1500://判断负极叠台搬运是否有片，有片的话放到纠偏台
	IF NOT DP_SinStepe THEN
		IF CA_CarryingPos1  THEN//负极搬运、叠片各轴在初始位
			IF arrCyCtrl[arrCyNo.ElectValveName.CaDTCarryingVacuum].Io.DIOnSwitch AND  Mach_Control.Ca_b.Ca_DPCarryingFalg THEN//正极再取片位且叠台搬运有片,把当前片放到纠偏台
				DP_Step0:=1550;
			ELSE
				DP_Step0:=3000;	
			END_IF
		ELSE
			IF (Ca_Step0=0 OR Ca_Step0=6666) AND (Ca_Step3=0 OR Ca_Step3=6666) AND Scan_TON[2].Q THEN
				Scan_TON[2].IN:=FALSE;		
				DP_Step0:=9994;
				DTPosError[2]:=TRUE;
			END_IF
		END_IF
	END_IF	
1550://纠偏台回初始位
	//纠偏平台X1移动至初始位
	IF NOT DP_SinStepe THEN
		IF arrAxisCtrl[AxiseNo.AxisName.CadeviationX1].Status.Homed  AND arrAxisCtrl[AxiseNo.AxisName.CadeviationX1].Status.NoMoving AND NOT  arrAxisCtrl[AxiseNo.AxisName.CadeviationX1].Status.Error THEN
			IF arrAxisCtrl[AxiseNo.AxisName.CadeviationX1].Cmd.arrbRealPoint[1] THEN
				arrAxisCtrl[AxiseNo.AxisName.CadeviationX1].Cmd.iGoSetPos:=0;
			ELSE
				arrAxisCtrl[AxiseNo.AxisName.CadeviationX1].Cmd.iGoSetPos:=1;
			END_IF					
		END_IF
		//纠偏平台X2移动至初始位
		IF arrAxisCtrl[AxiseNo.AxisName.CadeviationX2].Status.Homed  AND arrAxisCtrl[AxiseNo.AxisName.CadeviationX2].Status.NoMoving AND NOT  arrAxisCtrl[AxiseNo.AxisName.CadeviationX2].Status.Error THEN
			IF arrAxisCtrl[AxiseNo.AxisName.CadeviationX2].Cmd.arrbRealPoint[1] THEN
				arrAxisCtrl[AxiseNo.AxisName.CadeviationX2].Cmd.iGoSetPos:=0;
			ELSE
				arrAxisCtrl[AxiseNo.AxisName.CadeviationX2].Cmd.iGoSetPos:=1;
			END_IF					
		END_IF
		//纠偏平台X2移动至初始位
		IF arrAxisCtrl[AxiseNo.AxisName.CadeviationY].Status.Homed  AND arrAxisCtrl[AxiseNo.AxisName.CadeviationY].Status.NoMoving AND NOT  arrAxisCtrl[AxiseNo.AxisName.CadeviationY].Status.Error THEN
			IF arrAxisCtrl[AxiseNo.AxisName.CadeviationY].Cmd.arrbRealPoint[1] THEN
				arrAxisCtrl[AxiseNo.AxisName.CadeviationY].Cmd.iGoSetPos:=0;
			ELSE
				arrAxisCtrl[AxiseNo.AxisName.CadeviationY].Cmd.iGoSetPos:=1;
			END_IF					
		END_IF
		IF arrAxisCtrl[AxiseNo.AxisName.CadeviationX1].Cmd.arrbRealPoint[1] AND arrAxisCtrl[AxiseNo.AxisName.CadeviationX2].Cmd.arrbRealPoint[1] AND arrAxisCtrl[AxiseNo.AxisName.CadeviationY].Cmd.arrbRealPoint[1] THEN
			DT_SingeMode();//单步选择	
			DP_Step0:=1600;	
			DT_TON[5].IN:=FALSE;
		END_IF	
	END_IF
1600:
	IF NOT DP_SinStepe THEN
		IF arrAxisCtrl[AxiseNo.AxisName.CaDTCarryingUpDown].Cmd.arrbRealPoint[3] THEN
			arrAxisCtrl[AxiseNo.AxisName.CaDTCarryingUpDown].Cmd.iGoSetPos:=0;
			/// 吸盘破真空    纠偏台开真空
			arrCyCtrl[arrCyNo.ElectValveName.CaDTCarryingVacuum].Cmd.bON:=TRUE;	//负极叠台搬运升降真空	真空
			arrCyCtrl[arrCyNo.ElectValveName.CaDTCarryingVacuum].Cmd.bOFF:=FALSE;	//负极叠台搬运升降真空破真空								
			arrCyCtrl[arrCyNo.ElectValveName.CadeviationVacuum].Cmd.bON:=TRUE;	//负极纠偏台真空			
			arrCyCtrl[arrCyNo.ElectValveName.CadeviationVacuum].Cmd.bOFF:=FALSE;	//负极纠偏台真空	   
			DT_SingeMode();//单步选择	
			DP_Step0:=1650;
			DT_TON[5].IN:=TRUE;
		ELSE
			arrAxisCtrl[AxiseNo.AxisName.CaDTCarryingUpDown].Cmd.iGoSetPos:=3;//负极搬运升降2上升至凸轮耦合初始高度
		END_IF	
	END_IF
1650://叠台搬运极片放回纠偏台
	IF NOT DP_SinStepe THEN
		 IF DT_TON[5].Q THEN
				IF arrAxisCtrl[AxiseNo.AxisName.CaDTCarryingUpDown].Cmd.arrbRealPoint[4] THEN
					arrAxisCtrl[AxiseNo.AxisName.CaDTCarryingUpDown].Cmd.iGoSetPos:=0;
					/// 吸盘破真空    纠偏台开真空
					Mach_Control.Ca_b.Ca_deviationFalg:=TRUE;//复位纠偏平台有料标记
					Mach_Control.Ca_b.Ca_DPCarryingFalg:=FALSE;//负极搬运真空吸盘有料标记复位
					Par.stDT_date.Ca_MQ_Slice[8]:=Par.stDT_date.Ca_MQ_Slice[9];
					DT_SingeMode();//单步选择	
					DP_Step0:=1700;
					DT_TON[5].IN:=FALSE;
				ELSE
					arrAxisCtrl[AxiseNo.AxisName.CaDTCarryingUpDown].Cmd.iGoSetPos:=4;//负极搬运升降2上升至凸轮耦合初始高度
				END_IF		
	    END_IF	
	END_IF	
1700:
	DP_Step0:=3000;	
	


	
2000:		
	IF NOT DP_SinStepe THEN
		IF AN_CarryingPos1  THEN//正极搬运、叠片各轴在初始位										
			IF CA_CarryingPos2 THEN//负极在叠片位
				IF arrAxisCtrl[AxiseNo.AxisName.SEPTATLine].Cmd.arrbRealPoint[1]  THEN
					IF Mach_Control.DT_b.SinStepMode THEN//单步调试模式
						DP_SinStepe:=TRUE;
					ELSE
						DP_SinStepe:=FALSE;	
					END_IF
					DP_Step0:=2010;//
				ELSE
					Mach_Control.DT_b.Error[6]:=TRUE;//叠正极片凸轮耦合时，隔膜平移轴即不在负极叠片位，也不在正极叠片位报警
					DP_Step0:=9998;
				END_IF;
			ELSIF  CA_CarryingPos1  THEN //负极取片位
				IF arrAxisCtrl[AxiseNo.AxisName.SEPTATLine].Cmd.arrbRealPoint[1]  THEN
					IF Mach_Control.DT_b.SinStepMode THEN//单步调试模式
						DP_SinStepe:=TRUE;
					ELSE
						DP_SinStepe:=FALSE;	
					END_IF
					DP_Step0:=2030;//
				ELSIF arrAxisCtrl[AxiseNo.AxisName.SEPTATLine].Cmd.arrbRealPoint[2]  THEN
					IF Mach_Control.DT_b.SinStepMode THEN//单步调试模式
						DP_SinStepe:=TRUE;
					ELSE
						DP_SinStepe:=FALSE;	
					END_IF
					DP_Step0:=2050;//
				ELSE
					Mach_Control.DT_b.Error[6]:=TRUE;//叠正极片凸轮耦合时，隔膜平移轴即不在负极叠片位，也不在正极叠片位报警
					DP_Step0:=9999;
				END_IF;							
			ELSE
				Mach_Control.DT_b.Error[7]:=TRUE;//叠正极片凸轮耦合时，负极取片即不在取片位，也不在叠片位
				DP_Step0:=10000;
			END_IF
		ELSE
			Mach_Control.DT_b.Error[8]:=TRUE;//叠正极片凸轮耦合时，正极片不在取片位
			DP_Step0:=10001;
		END_IF
	END_IF		


2010://负极搬运、叠片各轴在初始位，隔膜平移轴负极叠片位、正极叠片在放极片初始位
	IF NOT DP_SinStepe THEN
		An_CanIn5:=TRUE;
		IF Mach_Control.DT_b.SinStepMode THEN//单步调试模式
				DP_SinStepe:=TRUE;
			ELSE
				DP_SinStepe:=FALSE;	
			END_IF
		DP_Step0:=2020;	
	END_IF	
2020:
	IF NOT DP_SinStepe THEN
		IF NOT An_CanIn5 THEN
			IF Mach_Control.DT_b.SinStepMode THEN//单步调试模式
				DP_SinStepe:=TRUE;
			ELSE
				DP_SinStepe:=FALSE;	
			END_IF	
			DP_Step0:=2070;
		ELSIF fbAnCamInCarryingLine.bError  OR fbAnCamInDTCarryingLine.bError OR fbAnCamInDTCarryingUpDown.bError OR 
			fbAnCamInCarryingWhirling.bError OR fbCaCamInCarryingLine2.bError OR 
			fbCaCamInDTCarryingUpDown.bError OR fbCamInGMBuffer.bError OR fbCamInGMDanserMove.bError OR fbCamInVirGMDriver.bError   OR
			fbCamInRightYDUpDown.bError OR fbCamInRightYDLine.bError  THEN
			An_CanIn5:=FALSE;
			Mach_Control.DT_b.Error[19]:=TRUE;//凸轮耦合报警
			DP_Step0:=10004;		
		END_IF
	END_IF		
2030://负极搬运、叠片各轴在初始位，隔膜平移轴负极叠片位、正极叠片在取极片位
	IF NOT DP_SinStepe THEN
		IF Mach_Control.DT_b.SinStepMode THEN//单步调试模式
			DP_SinStepe:=TRUE;
		ELSE
			DP_SinStepe:=FALSE;	
		END_IF
		An_CanIn6:=TRUE;
		DP_Step0:=2040;
	END_IF
2040:
	IF NOT DP_SinStepe THEN
		IF NOT An_CanIn6 THEN
			IF Mach_Control.DT_b.SinStepMode THEN//单步调试模式
				DP_SinStepe:=TRUE;
			ELSE
				DP_SinStepe:=FALSE;	
			END_IF
			DP_Step0:=2070;
		ELSIF fbAnCamInCarryingLine.bError OR fbAnCamInDTCarryingLine.bError OR
			fbAnCamInDTCarryingUpDown.bError OR fbAnCamInCarryingWhirling.bError OR fbCamInGMBuffer.bError OR
			fbCamInGMDanserMove.bError OR fbCamInVirGMDriver.bError  OR fbCamInRightYDUpDown.bError OR
			fbCamInRightYDLine.bError  THEN
			An_CanIn6:=FALSE;
			Mach_Control.DT_b.Error[19]:=TRUE;//凸轮耦合报警
			DP_Step0:=10002;									
		END_IF
	END_IF
2050://负极搬运、叠片各轴在初始位，隔膜平移轴正极叠片位、正极叠片在取极片位
	IF NOT DP_SinStepe THEN
		An_CanIn7:=TRUE;
		IF Mach_Control.DT_b.SinStepMode THEN//单步调试模式
				DP_SinStepe:=TRUE;
			ELSE
				DP_SinStepe:=FALSE;	
			END_IF
		DP_Step0:=2060;
	END_IF
2060:
	IF NOT DP_SinStepe THEN
			arrAxisCtrl[AxiseNo.VirAxisName.VirMain].Cmd	.bMoveAbs:=FALSE;	
			IF NOT An_CanIn7 THEN
				IF Mach_Control.DT_b.SinStepMode THEN//单步调试模式
					DP_SinStepe:=TRUE;
				ELSE
					DP_SinStepe:=FALSE;	
				END_IF
				DP_Step0:=2070;
			ELSIF fbAnCamInCarryingLine.bError OR fbAnCamInCarryingUpDown.bError OR fbAnCamInDTCarryingLine.bError OR fbAnCamInDTCarryingUpDown.bError OR 
				fbAnCamInCarryingWhirling.bError OR fbCamInRightYDUpDown.bError OR fbCamInRightYDLine.bError THEN
				An_CanIn7:=FALSE;
				Mach_Control.DT_b.Error[19]:=TRUE;//凸轮耦合报警
				DP_Step0:=10003;												
			END_IF
	END_IF	
	
2070://判断正极叠片搬运机械手上是否有极片

	IF NOT DP_SinStepe THEN
		VirMain_TON.IN:=FALSE;
		IF (NOT arrCyCtrl[arrCyNo.ElectValveName.AnDTCarryingVacuum].Io.DIOnSwitch AND NOT Mach_Control.An_b.An_DPCarryingFalg) OR Bnt_Blueflaging THEN	
			IF Mach_Control.DT_b.SinStepMode THEN//单步调试模式
				DP_SinStepe:=TRUE;
			ELSE
				DP_SinStepe:=FALSE;	
			END_IF
			DP_Step0:=2071;
		ELSE	
		  	Mach_Control.An_b.Error[28]:=TRUE; //正极叠片完空叠隔膜时，正极叠片搬运机械手真空有信号、标记有极片报警,请拿掉极片
		END_IF  
	END_IF

2071://主轴启动
	IF NOT DP_SinStepe THEN
		arrAxisCtrl[AxiseNo.VirAxisName.VirMain].Cmd	.bDynamitcsParSel:=2;	
		arrAxisPar[AxiseNo.VirAxisName.VirMain].fTagatTime:=VirMain_TagatTime;
		arrAxisCtrl[AxiseNo.VirAxisName.VirMain].Cmd	.fPositon_of_Abs:=360;
		arrAxisCtrl[AxiseNo.VirAxisName.VirMain].Cmd	.bMoveAbs:=TRUE;	
		//fbCaCamInCarryingUpDown2OutCamFlge:=FALSE;//负极升降2凸轮解耦标记										
		IF  arrAxis[AxiseNo.VirAxisName.VirMain].Status.Moving OR arrAxisCtrl[AxiseNo.VirAxisName.VirMain].Status.fActPos>=10  THEN
			VirMain_TON.IN:=FALSE;
			arrAxisCtrl[AxiseNo.VirAxisName.VirMain].Cmd	.bMoveAbs:=FALSE;	
			DP_Step0:=2080;	
		ELSE
			IF NOT VirMain_TON.Q THEN
				VirMain_TON.IN:=TRUE;
			ELSE
				VirMain_TON.IN:=FALSE;
				Mach_Control.DT_b.Error[22]:=TRUE;//主轴启动超时报警
				DP_Step0:=10006;	
			END_IF	
		END_IF	
	END_IF				
			
(*2080:
IF arrAxis[AxiseNo.VirAxisName.VirMain].NcToPlc.SetPos>=234 AND arrAxis[AxiseNo.VirAxisName.VirMain].NcToPlc.SetPos<=240 THEN
	arrCyCtrl[arrCyNo.ElectValveName.AnDTCarryingVacuum].Cmd.bOFF:=TRUE;//正极叠片搬运真空关
	arrCyCtrl[arrCyNo.ElectValveName.AnDTCarryingVacuumBark].Cmd.bON:=TRUE;//正极叠片搬运破真空开
	Mach_Control.An_b.An_DPCarryingFalg :=FALSE;//复位正极叠片搬运吸盘上有料标记																									
END_IF				
IF arrAxis[AxiseNo.VirAxisName.VirMain].NcToPlc.SetPos=360 AND  arrAxis[AxiseNo.VirAxisName.VirMain].Status.NotMoving  THEN
			Mach_Control.An_b.An_KDQuantited:=Mach_Control.An_b.An_KDQuantited +1;
			DP_Step1:=100;//解除耦合，主轴回零子程序
			arrAxisCtrl[AxiseNo.AxisName.DTUpDown].Cmd.fPosition_of_Rel:=-Par.stDT_date.SEPTA_Thickness;
			arrAxisPar[AxiseNo.AxisName.DTUpDown].fVelocity_of_Rel:=100;
			arrAxisCtrl[AxiseNo.AxisName.DTUpDown].Cmd.bMoveRel:=TRUE;
			DP_Step0:=0;
END_IF*)

3000:
	IF NOT DP_SinStepe THEN		
		Scan_TON[2].IN:=TRUE;	
		IF CA_CarryingPos1  THEN//负极搬运、叠片各轴在初始位
			Scan_TON[1].IN:=TRUE;	
			IF AN_CarryingPos2  THEN//正极在叠片位	
				IF arrAxisCtrl[AxiseNo.AxisName.SEPTATLine].Cmd.arrbRealPoint[2]   THEN													
					IF Mach_Control.DT_b.SinStepMode THEN//单步调试模式
						DP_SinStepe:=TRUE;
					ELSE
						DP_SinStepe:=FALSE;	
					END_IF												
					DP_Step0:=3010;//													
				ELSE
					Mach_Control.DT_b.Error[5]:=TRUE;//叠负极片凸轮耦合时，隔膜平移轴即不在负极叠片位，也不在正极叠片位报警
					DP_Step0:=9991;	
				END_IF;
			ELSIF AN_CarryingPos1  THEN//在取片位																		
				IF arrAxisCtrl[AxiseNo.AxisName.SEPTATLine].Cmd.arrbRealPoint[1]  THEN
					IF Mach_Control.DT_b.SinStepMode THEN//单步调试模式
						DP_SinStepe:=TRUE;
					ELSE
						DP_SinStepe:=FALSE;	
					END_IF											
					DP_Step0:=3030;//
				ELSIF arrAxisCtrl[AxiseNo.AxisName.SEPTATLine].Cmd.arrbRealPoint[2] THEN
					IF Mach_Control.DT_b.SinStepMode THEN//单步调试模式
						DP_SinStepe:=TRUE;
					ELSE
						DP_SinStepe:=FALSE;	
					END_IF											
					DP_Step0:=3050;//
				ELSE
					Mach_Control.DT_b.Error[5]:=TRUE;//叠负极片凸轮耦合时，隔膜平移轴即不在负极叠片位，也不在正极叠片位报警
					DP_Step0:=9992;	
				END_IF;							
			ELSIF Scan_TON[1].Q THEN
				Scan_TON[1].IN:=FALSE;	
				DP_Step0:=9993;
				DTPosError[4]:=TRUE;
			END_IF
		ELSE
			IF (Ca_Step0=0 OR Ca_Step0=6666) AND (Ca_Step3=0 OR Ca_Step3=6666) AND Scan_TON[2].Q THEN
				Scan_TON[2].IN:=FALSE;		
				DP_Step0:=9994;
				DTPosError[2]:=TRUE;
			END_IF
		END_IF
END_IF		

3010://负极搬运、叠片各轴在初始位，隔膜平移轴正极叠片位、正极叠片在放极片初始位
	IF NOT DP_SinStepe THEN
		Ca_CanIn5:=TRUE;
		IF Mach_Control.DT_b.SinStepMode THEN//单步调试模式
			DP_SinStepe:=TRUE;
		ELSE
			DP_SinStepe:=FALSE;	
		END_IF
		DP_Step0:=3020;	
	END_IF
3020:
	IF NOT DP_SinStepe THEN
		arrAxisCtrl[AxiseNo.VirAxisName.VirMain].Cmd	.bMoveAbs:=FALSE;	
		IF NOT Ca_CanIn5 THEN
			IF Mach_Control.DT_b.SinStepMode THEN//单步调试模式
				DP_SinStepe:=TRUE;
			ELSE
				DP_SinStepe:=FALSE;	
			END_IF
			DP_Step0:=3070;	
		ELSIF fbCaCamInCarryingLine2.bError OR  fbCaCamInDTCarryingLine.bError OR fbCaCamInDTCarryingUpDown.bError OR 
			fbCamInGMBuffer.bError OR fbCamInGMDanserMove.bError OR fbCamInVirGMDriver.bError OR fbAnCamInCarryingLine.bError OR 
			fbAnCamInDTCarryingLine.bError OR fbAnCamInCarryingWhirling.bError OR fbCamInLeftYDUpDown.bError OR fbCamInLeftYDLine.bError THEN
			Ca_CanIn5:=FALSE;
			Mach_Control.DT_b.Error[19]:=TRUE;//凸轮耦合报警
			DP_Step0:=9998;										
		END_IF
	END_IF
3030://负极搬运、叠片各轴在初始位，隔膜平移轴负极叠片位、正极叠片在取极片位
	IF NOT DP_SinStepe THEN
		Ca_CanIn6:=TRUE;
		IF Mach_Control.DT_b.SinStepMode THEN//单步调试模式
			DP_SinStepe:=TRUE;
		ELSE
			DP_SinStepe:=FALSE;	
		END_IF
		DP_Step0:=3040;
	END_IF
3040://判断凸轮耦合是否完成
	IF NOT DP_SinStepe THEN
		IF NOT Ca_CanIn6 THEN
			IF Mach_Control.DT_b.SinStepMode THEN//单步调试模式
				DP_SinStepe:=TRUE;
			ELSE
				DP_SinStepe:=FALSE;	
			END_IF
			DP_Step0:=3070;
		ELSIF  fbCaCamInCarryingLine2.bError OR fbCaCamInDTCarryingLine.bError OR 
			fbCaCamInDTCarryingUpDown.bError OR fbCamInLeftYDUpDown.bError OR 	fbCamInLeftYDLine.bError THEN										
			Ca_CanIn6:=FALSE;
			Mach_Control.DT_b.Error[19]:=TRUE;//凸轮耦合报警
			DP_Step0:=9995;		
		END_IF
	END_IF
3050://负极搬运、叠片各轴在初始位，隔膜平移轴正极叠片位、正极叠片在取极片位
	IF NOT DP_SinStepe THEN
		Ca_CanIn7:=TRUE;
		IF Mach_Control.DT_b.SinStepMode THEN//单步调试模式
			DP_SinStepe:=TRUE;
		ELSE
			DP_SinStepe:=FALSE;	
		END_IF
		DP_Step0:=3060;
	END_IF
3060:
	IF NOT DP_SinStepe THEN
			arrAxisCtrl[AxiseNo.VirAxisName.VirMain].Cmd	.bMoveAbs:=FALSE;	
			IF NOT Ca_CanIn7 THEN
				IF Mach_Control.DT_b.SinStepMode THEN//单步调试模式
					DP_SinStepe:=TRUE;
				ELSE
					DP_SinStepe:=FALSE;	
				END_IF																			
				DP_Step0:=3070;
			ELSIF fbCaCamInCarryingLine2.bError OR fbCaCamInDTCarryingLine.bError OR 
				fbCaCamInDTCarryingUpDown.bError OR fbCamInGMBuffer.bError OR fbCamInGMDanserMove.bError OR
				fbCamInVirGMDriver.bError OR fbCamInLeftYDUpDown.bError OR fbCamInLeftYDLine.bError  THEN
				Ca_CanIn7:=FALSE;
				Mach_Control.DT_b.Error[19]:=TRUE;//凸轮耦合报警
				DP_Step0:=9996;	
			END_IF
	END_IF

3070://判断负极叠片搬运机械手上是否有极片
	VirMain_TON.IN:=FALSE;
	DP_Step0:=3071;
	(*
	IF NOT DP_SinStepe THEN
		IF NOT arrCyCtrl[arrCyNo.ElectValveName.CaDTCarryingVacuum].Io.DIOnSwitch AND NOT Mach_Control.Ca_b.Ca_DPCarryingFalg  THEN	
			IF Mach_Control.DT_b.SinStepMode THEN//单步调试模式
				DP_SinStepe:=TRUE;
			ELSE
				DP_SinStepe:=FALSE;	
			END_IF
			DP_Step0:=3071;
		ELSE	
		  	Mach_Control.Ca_b.Error[28]:=TRUE; //负极叠片完空叠隔膜时，负极叠片搬运机械手真空检测有信号报警,请拿掉极片
		END_IF  
	END_IF	 
	*)
3071://主轴启动
	IF NOT DP_SinStepe THEN
		arrAxisCtrl[AxiseNo.VirAxisName.VirMain].Cmd	.bDynamitcsParSel:=2;
		arrAxisPar[AxiseNo.VirAxisName.VirMain].fTagatTime:=VirMain_TagatTime;
		arrAxisCtrl[AxiseNo.VirAxisName.VirMain].Cmd	.fPositon_of_Abs:=360;
		arrAxisCtrl[AxiseNo.VirAxisName.VirMain].Cmd	.bMoveAbs:=TRUE;	
		//fbCaCamInCarryingUpDown2OutCamFlge:=FALSE;//负极升降2凸轮解耦标记										
		IF  arrAxis[AxiseNo.VirAxisName.VirMain].Status.Moving OR arrAxisCtrl[AxiseNo.VirAxisName.VirMain].Status.fActPos>=10  THEN
			VirMain_TON.IN:=FALSE;
			arrAxisCtrl[AxiseNo.VirAxisName.VirMain].Cmd	.bMoveAbs:=FALSE;	
			DP_Step0:=3080;	
		ELSE
			IF NOT VirMain_TON.Q THEN
				VirMain_TON.IN:=TRUE;
			ELSE
				VirMain_TON.IN:=FALSE;
				Mach_Control.DT_b.Error[22]:=TRUE;//主轴启动超时报警
				DP_Step0:=10006;	
			END_IF	
		END_IF	
	END_IF	

END_CASE
END_IF


(**************************************************************************************电芯下料**************************************************************************************************************)
CASE DP_Step0 OF
2080:
IF arrAxis[AxiseNo.VirAxisName.VirMain].NcToPlc.SetPos>=234 AND arrAxis[AxiseNo.VirAxisName.VirMain].NcToPlc.SetPos<=240 THEN
	arrCyCtrl[arrCyNo.ElectValveName.AnDTCarryingVacuum].Cmd.bOFF:=FALSE;//正极叠片搬运升降真空关
     arrCyCtrl[arrCyNo.ElectValveName.AnDTCarryingVacuum].Cmd.bON:=TRUE;//正极叠片搬运升降真空关
	Mach_Control.An_b.An_DPCarryingFalg :=FALSE;//复位正极叠片搬运吸盘上有料标记																									
END_IF				
IF arrAxis[AxiseNo.VirAxisName.VirMain].NcToPlc.SetPos=360 AND  arrAxis[AxiseNo.VirAxisName.VirMain].Status.NotMoving  THEN
			Mach_Control.An_b.An_KDQuantited:=Mach_Control.An_b.An_KDQuantited +1;
			DP_Step1:=100;//解除耦合，主轴回零子程序
			arrAxisCtrl[AxiseNo.AxisName.DTUpDown].Cmd.fPosition_of_Rel:=-Par.stDT_date.SEPTA_Thickness;
			arrAxisPar[AxiseNo.AxisName.DTUpDown].fVelocity_of_Rel:=100;
			arrAxisCtrl[AxiseNo.AxisName.DTUpDown].Cmd.bMoveRel:=TRUE;
			DP_Step0:=0;
END_IF
	
(*2080:
	IF arrAxis[AxiseNo.VirAxisName.VirMain].NcToPlc.SetPos=360 AND  arrAxis[AxiseNo.VirAxisName.VirMain].Status.NotMoving  THEN
		Mach_Control.An_b.An_KDQuantited:=Mach_Control.An_b.An_KDQuantited +1;
		DPcount:=DPcount+1;	
		DP_Step1:=100;//解除耦合，主轴回零子程序
		arrAxisCtrl[AxiseNo.AxisName.DTUpDown].Cmd.fPosition_of_Rel:=-Par.stDT_date.SEPTA_Thickness;
		arrAxisPar[AxiseNo.AxisName.DTUpDown].fVelocity_of_Rel:=100;
		arrAxisCtrl[AxiseNo.AxisName.DTUpDown].Cmd.bMoveRel:=TRUE;
		DP_Step0:=0;
	END_IF*)


3080:

	IF arrAxis[AxiseNo.VirAxisName.VirMain].NcToPlc.SetPos=360 AND  arrAxis[AxiseNo.VirAxisName.VirMain].Status.NotMoving  THEN
		Mach_Control.Ca_b.Ca_KDQuantited:=Mach_Control.Ca_b.Ca_KDQuantited +1;
		DPcount:=DPcount+1;	
		DP_Step1:=100;//解除耦合，主轴回零子程序
		arrAxisCtrl[AxiseNo.AxisName.DTUpDown].Cmd.fPosition_of_Rel:=-Par.stDT_date.SEPTA_Thickness;
		arrAxisPar[AxiseNo.AxisName.DTUpDown].fVelocity_of_Rel:=100;
		arrAxisCtrl[AxiseNo.AxisName.DTUpDown].Cmd.bMoveRel:=TRUE;							
		DP_Step0:=0;
	END_IF		
END_CASE
END_ACTION

ACTION _01DT_Auto4:
IF Mach_Control.U.DT_iMode=1 THEN//在自动状态下
CASE DP_Step0 OF		
	6000://叠片完成，负极升降机械手回到安全位
			IF NOT DP_SinStepe THEN
						//负极取片2升降安全位
						IF arrAxisCtrl[AxiseNo.AxisName.CaCarryingUpDown2].Status.Homed AND arrAxisCtrl[AxiseNo.AxisName.CaCarryingUpDown2].Status.NoMoving AND 
							NOT arrAxisCtrl[AxiseNo.AxisName.CaCarryingUpDown2].Status.Error THEN
								IF arrAxisCtrl[AxiseNo.AxisName.CaCarryingUpDown2].Cmd.arrbRealPoint[4] THEN
										arrAxisCtrl[AxiseNo.AxisName.CaCarryingUpDown2].Cmd.iGoSetPos:=0;
								ELSE
									arrAxisCtrl[AxiseNo.AxisName.CaCarryingUpDown2].Cmd.iGoSetPos:=4;//负极搬运升降2移动至初始高度
								END_IF
						END_IF				
						//负极叠片取片升降等待位
						IF arrAxisCtrl[AxiseNo.AxisName.CaDTCarryingUpDown].Status.Homed AND arrAxisCtrl[AxiseNo.AxisName.CaDTCarryingUpDown].Status.NoMoving AND
							 NOT arrAxisCtrl[AxiseNo.AxisName.CaDTCarryingUpDown].Status.Error THEN
									IF arrAxisCtrl[AxiseNo.AxisName.CaDTCarryingUpDown].Cmd.arrbRealPoint[4] THEN
											arrAxisCtrl[AxiseNo.AxisName.CaDTCarryingUpDown].Cmd.iGoSetPos:=0;							
									ELSE
										arrAxisCtrl[AxiseNo.AxisName.CaDTCarryingUpDown].Cmd.iGoSetPos:=4;//负极叠片升降移动至等待高度
									END_IF
						END_IF
						
						IF 	arrAxisCtrl[AxiseNo.AxisName.CaCarryingUpDown2].Cmd.arrbRealPoint[4]  AND  arrAxisCtrl[AxiseNo.AxisName.CaCarryingUpDown2].Status.NoMoving AND 
								arrAxisCtrl[AxiseNo.AxisName.CaDTCarryingUpDown].Cmd.arrbRealPoint[4] 	AND arrAxisCtrl[AxiseNo.AxisName.CaDTCarryingUpDown].Status.NoMoving THEN
								IF Mach_Control.DT_b.SinStepMode THEN//单步调试模式
											DP_SinStepe:=TRUE;
								ELSE
											DP_SinStepe:=FALSE;	
								END_IF
								DP_Step0:=6010;
					END_IF
			END_IF
		6010://判断主轴是否停止、是否在初始位、是否有轴在耦合中
			IF NOT DP_SinStepe THEN
				IF CA_CarryingPos2 THEN
					IF arrAxisCtrl[AxiseNo.VirAxisName.VirMain].Status.NoMoving AND arrAxis[AxiseNo.VirAxisName.VirMain].NcToPlc.ActPos=0 AND NOT DT_AxiseCoupling THEN
						DT_SingeMode();//单步选择						
						DP_Step0:=6012;
					ELSE
						DP_Step1:=100;//调用主轴回初始位子程序
						DT_SingeMode();//单步选择							
						DP_Step0:=6011;
					END_IF
				ELSIF  CA_CarryingPos1 THEN
					DP_Step0:=6014;
				END_IF	
			END_IF
					
		6011://判断主轴的模长的当前位置是否为0
			IF NOT DP_SinStepe THEN
				IF DP_Step1=6666 AND arrAxisCtrl[AxiseNo.VirAxisName.VirMain].Status.NoMoving AND arrAxis[AxiseNo.VirAxisName.VirMain].NcToPlc.ActPos=0 AND NOT DT_AxiseCoupling THEN
					DT_SingeMode();//单步选择						
					DP_Step0:=6012;
				END_IF
			END_IF		

		6012:
			//负极送片搬运平移
				fbCaCamInCarryingLine2.ParCamIn.SlaveScaling:=-1;
				fbCaCamInCarryingLine2.bCamInExecute:=TRUE;								
		        fbCaCamInCarryingUpDown2.iTableSel:=3;    //20240528SJ
	            fbCaCamInCarryingUpDown2.bCamInExecute:=TRUE;		
				
			//负极叠台搬运平移
				fbCaCamInDTCarryingLine.ParCamIn.SlaveScaling:=-1;
				fbCaCamInDTCarryingLine.bCamInExecute:=TRUE;	
			    fbCaCamInDTCarryingUpDown.iTableSel:=3;   //20240528SJ
	            fbCaCamInDTCarryingUpDown.bCamInExecute:=TRUE;
				
			//负极叠片升降轴放片凸轮耦合
				//fbCaCamInDTCarryingUpDown.iTableSel:=2;
				//fbCaCamInDTCarryingUpDown.bCamInExecute:=TRUE;		
														  
			IF fbCaCamInCarryingLine2.bInSync AND fbCaCamInDTCarryingLine.bInSync AND  fbCaCamInCarryingUpDown2.bInSync AND fbCaCamInDTCarryingUpDown.bInSync   THEN   
				DT_SingeMode();//单步选择		
				DP_Step0:=6013;
			ELSIF fbCaCamInCarryingLine2.bError  OR  fbCaCamInDTCarryingLine.bError  OR 
                    fbCaCamInCarryingUpDown2.bError OR fbCaCamInDTCarryingUpDown.bError   THEN   
				Mach_Control.DT_b.Error[19]:=TRUE;//凸轮耦合报警
			END_IF	
		6074:	
			IF arrAxis[AxiseNo.VirAxisName.VirMain].NcToPlc.SetPos=360 AND  arrAxis[AxiseNo.VirAxisName.VirMain].Status.NotMoving THEN 
				DP_Step1:=100;
				DP_Step0:=6075;	
			END_IF
		  
		6075:  
			IF DP_Step1=6666 THEN	
				DP_Step0:=6014;						
			END_IF		
		  
		6014:
			IF arrAxisCtrl[AxiseNo.VirAxisName.VirMain].Status.NoMoving AND arrAxis[AxiseNo.VirAxisName.VirMain].NcToPlc.ActPos=0 AND NOT DT_AxiseCoupling 
				AND CA_CarryingPos1 THEN
				DP_Step0:=6015;	
			ELSIF  DT_AxiseCoupling THEN
				DP_Step1:=100;
				DP_Step0:=6075;	
			END_IF  
	(*
				IF NOT DP_SinStepe THEN
					//负极取片2平移取片位
											IF arrAxisCtrl[AxiseNo.AxisName.CaCarryingUpDown2].Cmd.arrbRealPoint[5] AND arrAxisCtrl[AxiseNo.AxisName.CaCarryingLine2].Status.Homed AND
												 arrAxisCtrl[AxiseNo.AxisName.CaCarryingLine2].Status.NoMoving AND NOT arrAxisCtrl[AxiseNo.AxisName.CaCarryingLine2].Status.Error THEN
													IF arrAxisCtrl[AxiseNo.AxisName.CaCarryingLine2].Cmd.arrbRealPoint[1] THEN
															arrAxisCtrl[AxiseNo.AxisName.CaCarryingLine2].Cmd.iGoSetPos:=0;					
													ELSE
														arrAxisCtrl[AxiseNo.AxisName.CaCarryingLine2].Cmd.iGoSetPos:=1;//负极搬运平移2移动至初始位取流水线上的极片
													END_IF
											END_IF
					//负极叠片平移取片位
										IF TailCurlSEPTA_SafePos  AND arrAxisCtrl[AxiseNo.AxisName.CaDTCarryingUpDown].Cmd.arrbRealPoint[4] AND arrAxisCtrl[AxiseNo.AxisName.CaDTCarryingLine].Status.Homed AND
											 arrAxisCtrl[AxiseNo.AxisName.CaDTCarryingLine].Status.NoMoving AND NOT arrAxisCtrl[AxiseNo.AxisName.CaDTCarryingLine].Status.Error THEN
												IF arrAxisCtrl[AxiseNo.AxisName.CaDTCarryingLine].Cmd.arrbRealPoint[1] THEN
														arrAxisCtrl[AxiseNo.AxisName.CaDTCarryingLine].Cmd.iGoSetPos:=0;
												ELSE
													arrAxisCtrl[AxiseNo.AxisName.CaDTCarryingLine].Cmd.iGoSetPos:=1;//负极叠片平移至初始位
												END_IF
										END_IF
										
										IF 	arrAxisCtrl[AxiseNo.AxisName.CaCarryingLine2].Cmd.arrbRealPoint[1] AND 	arrAxisCtrl[AxiseNo.AxisName.CaCarryingLine2].Status.NoMoving AND 
													arrAxisCtrl[AxiseNo.AxisName.CaDTCarryingLine].Cmd.arrbRealPoint[1] AND 	arrAxisCtrl[AxiseNo.AxisName.CaDTCarryingLine].Status.NoMoving THEN
													IF Mach_Control.DT_b.SinStepMode THEN//单步调试模式
																DP_SinStepe:=TRUE;
													ELSE
																DP_SinStepe:=FALSE;	
													END_IF
													DP_Step0:=6015;	
										//ELSIF  THEN											
										END_IF
				END_IF
	*)			
		6015:
			IF NOT DP_SinStepe THEN
					//负极叠片升降避让位
					IF arrAxisCtrl[AxiseNo.AxisName.CaDTCarryingUpDown].Status.Homed AND arrAxisCtrl[AxiseNo.AxisName.CaDTCarryingUpDown].Status.NoMoving AND
						 NOT arrAxisCtrl[AxiseNo.AxisName.CaDTCarryingUpDown].Status.Error THEN
						IF arrAxisCtrl[AxiseNo.AxisName.CaDTCarryingUpDown].Cmd.arrbRealPoint[5] THEN
								arrAxisCtrl[AxiseNo.AxisName.CaDTCarryingUpDown].Cmd.iGoSetPos:=0;							
						ELSE
							arrAxisCtrl[AxiseNo.AxisName.CaDTCarryingUpDown].Cmd.iGoSetPos:=5;//负极叠片升降移动至避让高度
						END_IF
					END_IF
					
					IF 	arrAxisCtrl[AxiseNo.AxisName.CaDTCarryingUpDown].Cmd.arrbRealPoint[5] 	AND arrAxisCtrl[AxiseNo.AxisName.CaDTCarryingUpDown].Status.NoMoving THEN
						IF Mach_Control.DT_b.SinStepMode THEN//单步调试模式
							DP_SinStepe:=TRUE;
						ELSE
							DP_SinStepe:=FALSE;	
						END_IF
						DP_Step0:=6016;
				END_IF
			END_IF
END_CASE
END_IF


CASE DP_Step0 OF
	6013:
		IF NOT DP_SinStepe THEN
			 arrAxisCtrl[AxiseNo.VirAxisName.VirMain].Cmd.bDynamitcsParSel:=2;	
			 arrAxisPar[AxiseNo.VirAxisName.VirMain].fTagatTime:=VirMain_TagatTime;
			 arrAxisCtrl[AxiseNo.VirAxisName.VirMain].Cmd.fPositon_of_Abs:=360;
			 arrAxisCtrl[AxiseNo.VirAxisName.VirMain].Cmd.bMoveAbs:=TRUE;			
			IF  arrAxis[AxiseNo.VirAxisName.VirMain].Status.Moving OR arrAxisCtrl[AxiseNo.VirAxisName.VirMain].Status.fActPos>=5  THEN		
				arrAxisCtrl[AxiseNo.VirAxisName.VirMain].Cmd.bMoveAbs:=FALSE;
				Ca_TON[2].IN:=FALSE;                               	
				DP_Step0:=6074;	
				//Ca_StandbyStep1:=300;  //取消调用负极送片搬运取流水线极片
				//Ca_StandbyStep5:=400;
			ELSE
				IF NOT Ca_TON[2].Q THEN
					Ca_TON[2].IN:=TRUE;
				ELSE
				Ca_TON[2].IN:=FALSE;
					Mach_Control.DT_b.Error[22]:=TRUE;//主轴启动超时报警
					arrAxisCtrl[AxiseNo.VirAxisName.VirMain].Cmd	.bMoveAbs:=FALSE;	
				END_IF
			END_IF	
		END_IF	
					
	6016://纠偏平台回原
		 IF arrAxisCtrl[AxiseNo.AxisName.AnDTCarryingUpDown].Cmd.arrbRealPoint[4] AND arrAxisCtrl[AxiseNo.AxisName.CaDTCarryingUpDown].Cmd.arrbRealPoint[5]  THEN
			 DP_Step11:=100;//正极纠偏平台回原
			 DP_Step12:=100;//负极纠偏平台回原
			 DP_Step0:=6020;
		 END_IF


	6020:
				IF Mach_Control.DT_b.DT_Oerhang_Z<>2 OR   Mach_Control.DT_b.DT_Overhang THEN
					CellMemory[Mach_Control.DT_b.DT_Memory].Hough:=1;
					DP_Step0:=6025;
					NN:=0;
				ELSE 
					CellMemory[Mach_Control.DT_b.DT_Memory].Hough:=2;
					DP_Step0:=6024;
				END_IF
				
	6024:
				NN:=NN+1;
				DP_Step0:=6025;			
																
	6025:
			Mach_Control.DT_b.DT_amount:=Mach_Control.DT_b.DT_amount+1;
			CellMemory[Mach_Control.DT_b.DT_Memory].Cell:=TRUE;	
			CellMemory[Mach_Control.DT_b.DT_Memory].DT_station_No:=Mach_Control.DT_b.DT_No;
			CellMemory[Mach_Control.DT_b.DT_Memory].DT_speed:=Par.stDT_date.SinglePosTime;
			CellMemory[Mach_Control.DT_b.DT_Memory].An_Quantity:=Mach_Control.An_b.An_Quantited;
			CellMemory[Mach_Control.DT_b.DT_Memory].Ca_Quantity:=Mach_Control.Ca_b.Ca_Quantited;
			//CellMemory[Mach_Control.DT_b.DT_Memory].DiaphragmUnwindingTension:=LIMIT(150,Mach_Control.DT_b.DiaphragmUnwindingTension,250);	
            // CellMemory[Mach_Control.DT_b.DT_Memory].DiaphragmUnwindingTension:=CellMemory[Mach_Control.DT_b.DT_Memory].Chipdata[210].GMlapTen;				
			//CellMemory[Mach_Control.DT_b.DT_Memory].DiaphragmUnwindingTension_max:=ABS(Mach_Control.DT_b.DiaphragmUnwindingTension+10);	
			//CellMemory[Mach_Control.DT_b.DT_Memory].DiaphragmUnwindingTension_min:=ABS(Mach_Control.DT_b.DiaphragmUnwindingTension-4);	
			//CellMemory[Mach_Control.DT_b.DT_Memory].DiaphragmUnwindingTension_ave:=ABS(Mach_Control.DT_b.DiaphragmUnwindingTension+5);	
			//[Mach_Control.DT_b.DT_Memory].DiaphragmUnwindingTension_set:=ABS(Mach_Control.DT_b.DiaphragmUnwindingTension);
	
            CellMemory[Mach_Control.DT_b.DT_Memory].DiaphragmUnwindingTension:=LIMIT(150,CellMemory[Mach_Control.DT_b.DT_Memory].Chipdata[210].GMlapTen,250);				
			CellMemory[Mach_Control.DT_b.DT_Memory].DiaphragmUnwindingTension_max:=LIMIT(150,CellMemory[Mach_Control.DT_b.DT_Memory].Chipdata[210].GMlapTen+10,250);	
			CellMemory[Mach_Control.DT_b.DT_Memory].DiaphragmUnwindingTension_min:=LIMIT(150,CellMemory[Mach_Control.DT_b.DT_Memory].Chipdata[210].GMlapTen-4,250);	
			CellMemory[Mach_Control.DT_b.DT_Memory].DiaphragmUnwindingTension_ave:=LIMIT(150,CellMemory[Mach_Control.DT_b.DT_Memory].Chipdata[210].GMlapTen+5,250);	
			CellMemory[Mach_Control.DT_b.DT_Memory].DiaphragmUnwindingTension_set:=LIMIT(150,CellMemory[Mach_Control.DT_b.DT_Memory].Chipdata[210].GMlapTen,250);	
			
			CellMemory[Mach_Control.DT_b.DT_Memory].Put_Time :=Mach_Control.DT_b.Put_time;
			CellMemory[Mach_Control.DT_b.DT_Memory].Machine_No:=Mach_Control.DT_b.Machine_No;
			CellMemory[Mach_Control.DT_b.DT_Memory].Cell_CCD_No:=CCD.Over.Finish.stCellNo;
			CellMemory[Mach_Control.DT_b.DT_Memory].BlueGlue:=1;
			
			CellMemory[Mach_Control.DT_b.DT_Memory].An_stuff_No:=Par.stDT_date.An_stuff_No;
			CellMemory[Mach_Control.DT_b.DT_Memory].Ca_stuff_No:=Par.stDT_date.Ca_stuff_No;
			CellMemory[Mach_Control.DT_b.DT_Memory].Diaphragm_No:=Par.stDT_date.Diaphragm_No;
			CellMemory[Mach_Control.DT_b.DT_Memory].PostiveCode:=CellMemory[Mach_Control.DT_b.DT_Memory].An_MQ_Slice[Mach_Control.An_b.An_Quantited].Code;//正极片条码
			CellMemory[Mach_Control.DT_b.DT_Memory].NegativeCode:=CellMemory[Mach_Control.DT_b.DT_Memory].Ca_MQ_Slice[Mach_Control.Ca_b.Ca_Quantited].Code;//负极片条码
		
		    CellMemory[Mach_Control.DT_b.DT_Memory].LYDLineinitPos:=arrAxisPar[AxiseNo.AxisName.LeftYDLine].arrTargetPoint[1];
			CellMemory[Mach_Control.DT_b.DT_Memory].LYDLineOpenPos :=arrAxisPar[AxiseNo.AxisName.LeftYDLine].arrTargetPoint[2];
			CellMemory[Mach_Control.DT_b.DT_Memory].LYDLinepressL :=arrAxisPar[AxiseNo.AxisName.LeftYDLine].arrTargetPoint[12];
			CellMemory[Mach_Control.DT_b.DT_Memory].RYDLineinitPos:=arrAxisPar[AxiseNo.AxisName.RightYDLine].arrTargetPoint[1];
			CellMemory[Mach_Control.DT_b.DT_Memory].RYDLineOpenPos :=arrAxisPar[AxiseNo.AxisName.RightYDLine].arrTargetPoint[2];
			CellMemory[Mach_Control.DT_b.DT_Memory].RYDLinepressL :=arrAxisPar[AxiseNo.AxisName.RightYDLine].arrTargetPoint[12];
			CellMemory[Mach_Control.DT_b.DT_Memory].LYDUpDowninitPos:=arrAxisPar[AxiseNo.AxisName.LeftYDUpDown].arrTargetPoint[1];
			CellMemory[Mach_Control.DT_b.DT_Memory].LYDUpDownOpenPos :=arrAxisPar[AxiseNo.AxisName.LeftYDUpDown].arrTargetPoint[2];
			CellMemory[Mach_Control.DT_b.DT_Memory].LYDUpDownOpenH:=arrAxisPar[AxiseNo.AxisName.LeftYDUpDown].arrTargetPoint[11];
			CellMemory[Mach_Control.DT_b.DT_Memory].LYDUpDownKnifeH:=arrAxisPar[AxiseNo.AxisName.LeftYDUpDown].arrTargetPoint[12];
			CellMemory[Mach_Control.DT_b.DT_Memory].RYDUpDowninitPos :=arrAxisPar[AxiseNo.AxisName.RightYDUpDown].arrTargetPoint[1];
			CellMemory[Mach_Control.DT_b.DT_Memory].RYDUpDownOpenPos :=arrAxisPar[AxiseNo.AxisName.RightYDUpDown].arrTargetPoint[2];
			CellMemory[Mach_Control.DT_b.DT_Memory].RYDUpDownOpenH:=arrAxisPar[AxiseNo.AxisName.RightYDUpDown].arrTargetPoint[11];
			CellMemory[Mach_Control.DT_b.DT_Memory].RYDUpDownKnifeH:=arrAxisPar[AxiseNo.AxisName.RightYDUpDown].arrTargetPoint[12];
			CellMemory[Mach_Control.DT_b.DT_Memory].DTandescendh:=Par.stDT_date.An_Thickness+Par.stDT_date.SEPTA_Thickness+Par.stDT_date.Pole_ThicknessCom;
			CellMemory[Mach_Control.DT_b.DT_Memory].DTcadescendh:=Par.stDT_date.Ca_Thickness+Par.stDT_date.SEPTA_Thickness+Par.stDT_date.Pole_ThicknessCom;
		
			
			IF Mach_Control.DT_b.DT_DebugMode THEN
			   CellMemory[Mach_Control.DT_b.DT_Memory].DTDebugMode:=TRUE;
			END_IF
			
			IF Mach_Control.DT_b.Overhang_TF THEN
			CellMemory[Mach_Control.DT_b.DT_Memory].Overhang_TF:=TRUE;
			ELSE
			CellMemory[Mach_Control.DT_b.DT_Memory].Overhang_TF:=FALSE;	
			END_IF
			DP_Step0:=6030;	

					
	6030:			
				Mach_Control.DT_b.Overhang_TF:=FALSE;	
				Mach_Control.DT_b.OffloadRequest:=TRUE;//叠电芯完成，请求下电芯
				DP_Step0:=6040;	
	6040://
		IF Mach_Control.DT_b.OffloadDone THEN
			bFirstFoldFinish[1]:=FALSE;//首层隔膜空叠
			bFirstFoldFinish[2]:=FALSE;//正常电芯空叠隔膜
			bFirstFoldFinish[3]:=FALSE;//接带、黄标空叠隔膜
			bEmptyFoldMark[1]:=FALSE;//进入空叠流程
			bEmptyFoldMark[2]:=FALSE;//进入空叠流程
			bEmptyFoldMark[3]:=FALSE;//进入空叠流程	
			Mach_Control.An_b.An_FirstFoldCnt:=0;
			Mach_Control.Ca_b.Ca_FirstFoldCnt:=0;
			Mach_Control.DT_b.OffloadRequest:=FALSE;//叠电芯完成，请求下电芯
			Mach_Control.An_b.An_Quantited:=0;
			Mach_Control.Ca_b.Ca_Quantited:=0;
			Mach_Control.An_b.An_KDQuantited :=0;
			Mach_Control.Ca_b.Ca_KDQuantited:=0;
			Mach_Control.DT_b.OffloadDone:=FALSE;
			OversequelNG:=FALSE;	
			DP_Step0:=6041;	
		END_IF

	6041://负极叠台升降、取片升降到等待高度等待耦合
		IF arrAxisCtrl[AxiseNo.AxisName.CaDTCarryingUpDown].Cmd.arrbRealPoint[4] THEN
			arrAxisCtrl[AxiseNo.AxisName.CaDTCarryingUpDown].Cmd.iGoSetPos:=0;				
		ELSE
			arrAxisCtrl[AxiseNo.AxisName.CaDTCarryingUpDown].Cmd.iGoSetPos:=4;//负极叠片升降移动至取片位
		END_IF
		IF arrAxisCtrl[AxiseNo.AxisName.CaCarryingUpDown2].Cmd.arrbRealPoint[4] THEN
			arrAxisCtrl[AxiseNo.AxisName.CaCarryingUpDown2].Cmd.iGoSetPos:=0;				
		ELSE
			arrAxisCtrl[AxiseNo.AxisName.CaCarryingUpDown2].Cmd.iGoSetPos:=4;//负极叠片升降移动至取片位
		END_IF
		IF  arrAxisCtrl[AxiseNo.AxisName.CaDTCarryingUpDown].Cmd.arrbRealPoint[4] AND arrAxisCtrl[AxiseNo.AxisName.CaCarryingUpDown2].Cmd.arrbRealPoint[4] THEN
			DP_Step0:=6042;
		END_IF
	
	6042://	等待纠偏平台回原完成		
			IF DP_Step11=6666 AND DP_Step12=6666 THEN
			   DP_Step0:=0;
			END_IF															
END_CASE
END_ACTION

ACTION _01DT_Auto5:

//
IF Ca_CanIn1 THEN  //OK
//负到正_负极搬运平移2轴凸轮耦合
	fbCaCamInCarryingLine2.ParCamIn.SlaveScaling:=1;
	fbCaCamInCarryingLine2.bCamInExecute:=TRUE;
//负到正_负极搬运升降2轴放片凸轮耦合
	fbCaCamInCarryingUpDown2.iTableSel:=2;
	fbCaCamInCarryingUpDown2.bCamInExecute:=TRUE;
//负到正_负极叠片平移轴凸轮耦合
	fbCaCamInDTCarryingLine.ParCamIn.SlaveScaling:=1;
	fbCaCamInDTCarryingLine.bCamInExecute:=TRUE;
//负到正_负极叠片升降轴放片凸轮耦合
	fbCaCamInDTCarryingUpDown.iTableSel:=2;
	fbCaCamInDTCarryingUpDown.bCamInExecute:=TRUE;
//叠台左压刀升降凸轮耦合
	//fbCamInLeftYDUpDown.bCamInExecute:=TRUE;
//叠台左压刀开合凸轮耦合
	//fbCamInLeftYDLine.bCamInExecute:=TRUE;
IF arrAxisCtrl[AxiseNo.AxisName.LeftYDLine].Cmd.arrbRealPoint[1] THEN
	fbCamInLeftYDUpDown.iTableSel:=1;
	fbCamInLeftYDLine.iTableSel:=1;
	fbCamInLeftYDUpDown.bCamInExecute:=TRUE;
	fbCamInLeftYDLine.bCamInExecute:=TRUE;	
ELSIF arrAxisCtrl[AxiseNo.AxisName.LeftYDLine].Cmd.arrbRealPoint[2] THEN	
	fbCamInLeftYDUpDown.iTableSel:=2;
	fbCamInLeftYDLine.iTableSel:=2;
	fbCamInLeftYDUpDown.bCamInExecute:=TRUE;
	fbCamInLeftYDLine.bCamInExecute:=TRUE;		
END_IF
//判断凸轮耦合是否完成
	IF 	fbCaCamInCarryingLine2.bInSync AND fbCaCamInCarryingUpDown2	.bInSync AND 	fbCaCamInDTCarryingLine.bInSync AND 	fbCaCamInDTCarryingUpDown.bInSync AND 
		fbCamInLeftYDUpDown.bInSync AND fbCamInLeftYDLine.bInSync 	 THEN
		Ca_CanIn1:=FALSE;
		//DP_Step0:=141;
	END_IF	
END_IF
//
IF Ca_CanIn2 THEN //OK
//负到正_负极搬运平移2轴凸轮耦合
	fbCaCamInCarryingLine2.ParCamIn.SlaveScaling:=1;
	fbCaCamInCarryingLine2.bCamInExecute:=TRUE;						
//负到正_负极搬运升降2轴放片凸轮耦合
	fbCaCamInCarryingUpDown2.iTableSel:=2;
	fbCaCamInCarryingUpDown2.bCamInExecute:=TRUE;
//负到正_负极叠片平移轴凸轮耦合
	fbCaCamInDTCarryingLine.ParCamIn.SlaveScaling:=1;
	fbCaCamInDTCarryingLine.bCamInExecute:=TRUE;						
//负到正_负极叠片升降轴放片凸轮耦合
	fbCaCamInDTCarryingUpDown.iTableSel:=2;
	fbCaCamInDTCarryingUpDown.bCamInExecute:=TRUE;
//负到正_缓存轴凸轮耦合	
	fbCamInGMBuffer.iTableSel:=2;
	fbCamInGMBuffer.bCamInExecute:=TRUE;
//负到正_隔膜平移轴凸轮耦合
	fbCamInGMDanserMove.iTableSel:=2;
	fbCamInGMDanserMove.bCamInExecute:=TRUE;

//负到正_放卷虚轴凸轮耦合
	fbCamInVirGMDriver.iTableSel:=2;
	fbCamInVirGMDriver.bCamInExecute:=TRUE;
//叠台左压刀升降凸轮耦合
	//fbCamInLeftYDUpDown.bCamInExecute:=TRUE;
//叠台左压刀开合凸轮耦合
	//fbCamInLeftYDLine.bCamInExecute:=TRUE;	
IF arrAxisCtrl[AxiseNo.AxisName.LeftYDLine].Cmd.arrbRealPoint[1] THEN
	fbCamInLeftYDUpDown.iTableSel:=1;
	fbCamInLeftYDLine.iTableSel:=1;
	fbCamInLeftYDUpDown.bCamInExecute:=TRUE;
	fbCamInLeftYDLine.bCamInExecute:=TRUE;	
ELSIF arrAxisCtrl[AxiseNo.AxisName.LeftYDLine].Cmd.arrbRealPoint[2] THEN	
	fbCamInLeftYDUpDown.iTableSel:=2;
	fbCamInLeftYDLine.iTableSel:=2;
	fbCamInLeftYDUpDown.bCamInExecute:=TRUE;
	fbCamInLeftYDLine.bCamInExecute:=TRUE;		
END_IF
					
//判断凸轮耦合是否完成
	IF fbCaCamInCarryingLine2.bInSync AND fbCaCamInCarryingUpDown2.bInSync AND fbCaCamInDTCarryingLine.bInSync AND
		fbCaCamInDTCarryingUpDown.bInSync AND fbCamInGMBuffer.bInSync AND fbCamInGMDanserMove.bInSync AND 
		fbCamInVirGMDriver.bInSync AND fbCamInLeftYDUpDown.bInSync AND fbCamInLeftYDLine.bInSync    THEN								
		Ca_CanIn2:=FALSE;
		//DP_Step0:=141;
	END_IF
END_IF
//
IF Ca_CanIn3 THEN    //OK
//负到正_负极搬运平移2轴凸轮耦合
	fbCaCamInCarryingLine2.ParCamIn.SlaveScaling:=1;
	fbCaCamInCarryingLine2.bCamInExecute:=TRUE;									
//负到正_负极搬运升降2轴放片凸轮耦合
	fbCaCamInCarryingUpDown2.iTableSel:=2;
	fbCaCamInCarryingUpDown2.bCamInExecute:=TRUE;
//负到正_负极叠片平移轴凸轮耦合
	fbCaCamInDTCarryingLine.ParCamIn.SlaveScaling:=1;
	fbCaCamInDTCarryingLine.bCamInExecute:=TRUE;							
//负到正_负极叠片升降轴放片凸轮耦合
	fbCaCamInDTCarryingUpDown.iTableSel:=2;
	fbCaCamInDTCarryingUpDown.bCamInExecute:=TRUE;						
//负到正_正极搬运平移轴凸轮耦合
	fbAnCamInCarryingLine.ParCamIn.SlaveScaling:=-1;
	fbAnCamInCarryingLine.bCamInExecute:=TRUE;
//负到正_正极搬运升降轴取片凸轮耦合	
	fbAnCamInCarryingUpDown.iTableSel:=1;	
	fbAnCamInCarryingUpDown.bCamInExecute:=TRUE;
//负到正_正极叠片平移轴凸轮耦合
	fbAnCamInDTCarryingLine.ParCamIn.SlaveScaling:=-1;
	fbAnCamInDTCarryingLine.bCamInExecute:=TRUE;
//负到正_正极叠片升降轴取片凸轮耦合
	fbAnCamInDTCarryingUpDown.iTableSel:=1;
	fbAnCamInDTCarryingUpDown.bCamInExecute:=TRUE;
//负到正_正极搬运旋转轴凸轮耦合	
	fbAnCamInCarryingWhirling.ParCamIn.SlaveScaling:=-1;
	fbAnCamInCarryingWhirling.bCamInExecute:=TRUE;
//叠台左压刀升降凸轮耦合
	//fbCamInLeftYDUpDown.bCamInExecute:=TRUE;
//叠台左压刀开合凸轮耦合
	//fbCamInLeftYDLine.bCamInExecute:=TRUE;
IF arrAxisCtrl[AxiseNo.AxisName.LeftYDLine].Cmd.arrbRealPoint[1] THEN
	fbCamInLeftYDUpDown.iTableSel:=1;
	fbCamInLeftYDLine.iTableSel:=1;
	fbCamInLeftYDUpDown.bCamInExecute:=TRUE;
	fbCamInLeftYDLine.bCamInExecute:=TRUE;	
ELSIF arrAxisCtrl[AxiseNo.AxisName.LeftYDLine].Cmd.arrbRealPoint[2] THEN	
	fbCamInLeftYDUpDown.iTableSel:=2;
	fbCamInLeftYDLine.iTableSel:=2;
	fbCamInLeftYDUpDown.bCamInExecute:=TRUE;
	fbCamInLeftYDLine.bCamInExecute:=TRUE;		
END_IF									
//	判断凸轮耦合是否完成
	IF fbCaCamInCarryingLine2.bInSync AND fbCaCamInCarryingUpDown2.bInSync AND fbCaCamInDTCarryingLine.bInSync AND fbCaCamInDTCarryingUpDown.bInSync AND 
		fbAnCamInCarryingLine.bInSync AND fbAnCamInCarryingUpDown.bInSync AND fbAnCamInDTCarryingLine.bInSync AND fbAnCamInDTCarryingUpDown.bInSync AND
		fbAnCamInCarryingWhirling.bInSync AND fbCamInLeftYDUpDown.bInSync AND fbCamInLeftYDLine.bInSync THEN
		Ca_CanIn3:=FALSE;
		//DP_Step0:=161;
	END_IF				
END_IF

//
IF Ca_CanIn4 THEN    //OK
//负到正_负极搬运平移2轴凸轮耦合
	fbCaCamInCarryingLine2.ParCamIn.SlaveScaling:=1;
	fbCaCamInCarryingLine2.bCamInExecute:=TRUE;							
//负到正_负极搬运升降2轴放片凸轮耦合
	fbCaCamInCarryingUpDown2.iTableSel:=2;
	fbCaCamInCarryingUpDown2.bCamInExecute:=TRUE;					
//负到正_负极叠片平移轴凸轮耦合
	fbCaCamInDTCarryingLine.ParCamIn.SlaveScaling:=1;
	fbCaCamInDTCarryingLine.bCamInExecute:=TRUE;							
//负到正_负极叠片升降轴放片凸轮耦合
	fbCaCamInDTCarryingUpDown.iTableSel:=2;
	fbCaCamInDTCarryingUpDown.bCamInExecute:=TRUE;		
//负到正_缓存轴凸轮耦合
	fbCamInGMBuffer.iTableSel:=2;
	fbCamInGMBuffer.bCamInExecute:=TRUE;					
//负到正_隔膜平移轴凸轮耦合
	fbCamInGMDanserMove.iTableSel:=2;
	fbCamInGMDanserMove.bCamInExecute:=TRUE;

	
//负到正_放卷虚轴凸轮耦合		
	fbCamInVirGMDriver.iTableSel:=2;
	fbCamInVirGMDriver.bCamInExecute:=TRUE;		
//负到正_正极搬运平移轴凸轮耦合	
	fbAnCamInCarryingLine.ParCamIn.SlaveScaling:=-1;
	fbAnCamInCarryingLine.bCamInExecute:=TRUE;															
//负到正_正极搬运升降轴取片凸轮耦合
	IF NOT DP_CheseCam THEN//???????????????
		fbAnCamInCarryingUpDown.iTableSel:=3;  //20240528SJ
		fbAnCamInCarryingUpDown.bCamInExecute:=TRUE;
	ELSE
		fbAnCamInCarryingUpDown.iTableSel:=3;  //20240528SJ
		fbAnCamInCarryingUpDown.bCamInExecute:=TRUE;		
	END_IF
	
//负到正_正极叠片平移轴凸轮耦合
	fbAnCamInDTCarryingLine.ParCamIn.SlaveScaling:=-1;
	fbAnCamInDTCarryingLine.bCamInExecute:=TRUE;	
//负到正_正极叠片升降轴取片凸轮耦合
IF NOT DP_CheseCam AND iAnCamInSel2=1 THEN
	fbAnCamInDTCarryingUpDown.iTableSel:=1;
	fbAnCamInDTCarryingUpDown.bCamInExecute:=TRUE;
ELSE
	fbAnCamInDTCarryingUpDown.iTableSel:=3;//20240528SJ
	fbAnCamInDTCarryingUpDown.bCamInExecute:=TRUE;	
END_IF

//负到正_正极搬运旋转轴凸轮耦合
	fbAnCamInCarryingWhirling.ParCamIn.SlaveScaling:=-1;
	fbAnCamInCarryingWhirling.bCamInExecute:=TRUE;
//叠台左压刀升降凸轮耦合
	//fbCamInLeftYDUpDown.bCamInExecute:=TRUE;
//叠台左压刀开合凸轮耦合
	//fbCamInLeftYDLine.bCamInExecute:=TRUE;	
IF arrAxisCtrl[AxiseNo.AxisName.LeftYDLine].Cmd.arrbRealPoint[1] THEN
	fbCamInLeftYDUpDown.iTableSel:=1;
	fbCamInLeftYDLine.iTableSel:=1;
	fbCamInLeftYDUpDown.bCamInExecute:=TRUE;
	fbCamInLeftYDLine.bCamInExecute:=TRUE;	
ELSIF arrAxisCtrl[AxiseNo.AxisName.LeftYDLine].Cmd.arrbRealPoint[2] THEN	
	fbCamInLeftYDUpDown.iTableSel:=2;
	fbCamInLeftYDLine.iTableSel:=2;
	fbCamInLeftYDUpDown.bCamInExecute:=TRUE;
	fbCamInLeftYDLine.bCamInExecute:=TRUE;		
END_IF				
//判断凸轮是否耦合完成
	IF fbCaCamInCarryingLine2.bInSync AND fbCaCamInCarryingUpDown2.bInSync AND fbCaCamInDTCarryingLine.bInSync AND  fbCaCamInDTCarryingUpDown.bInSync AND
	   fbCamInGMBuffer.bInSync AND fbCamInGMDanserMove.bInSync AND  fbCamInVirGMDriver.bInSync AND
		 fbAnCamInCarryingLine.bInSync AND fbAnCamInCarryingUpDown.bInSync AND  fbAnCamInCarryingWhirling.bInSync AND
		 fbAnCamInDTCarryingLine.bInSync AND ((fbAnCamInDTCarryingUpDown.bInSync AND  iAnCamInSel2=1 ) OR  (iAnCamInSel2=2 AND fbAnCamInDTCarryingUpDown.bInSync ) )AND
          fbCamInLeftYDUpDown.bInSync AND fbCamInLeftYDLine.bInSync  AND NOT DP_CheseCam THEN
		Ca_CanIn4:=FALSE;
		//DP_Step0:=161;
	ELSIF fbCaCamInCarryingLine2.bInSync AND fbCaCamInCarryingUpDown2.bInSync AND fbCaCamInDTCarryingLine.bInSync AND fbCaCamInDTCarryingUpDown.bInSync AND
		 fbCamInGMBuffer.bInSync AND fbCamInGMDanserMove.bInSync AND  fbCamInVirGMDriver.bInSync AND
		fbAnCamInCarryingLine.bInSync AND fbAnCamInCarryingUpDown.bInSync AND  fbAnCamInCarryingWhirling.bInSync AND  
       fbAnCamInDTCarryingLine.bInSync AND fbAnCamInDTCarryingUpDown.bInSync AND
        fbCamInLeftYDUpDown.bInSync AND fbCamInLeftYDLine.bInSync  AND DP_CheseCam THEN
		Ca_CanIn4:=FALSE;
		//DP_Step0:=161;
	END_IF		
END_IF


//
IF Ca_CanIn5 THEN   //OK
//负到正_负极搬运平移2轴凸轮耦合
	fbCaCamInCarryingLine2.ParCamIn.SlaveScaling:=1;
	fbCaCamInCarryingLine2.bCamInExecute:=TRUE;							
//负到正_负极搬运升降2轴放片凸轮耦合
	fbCaCamInCarryingUpDown2.iTableSel:=3;    //20240528SJ
	fbCaCamInCarryingUpDown2.bCamInExecute:=TRUE;					
//负到正_负极叠片平移轴凸轮耦合
	fbCaCamInDTCarryingLine.ParCamIn.SlaveScaling:=1;
	fbCaCamInDTCarryingLine.bCamInExecute:=TRUE;							
//负到正_负极叠片升降轴放片凸轮耦合
	
	fbCaCamInDTCarryingUpDown.iTableSel:=2;
	fbCaCamInDTCarryingUpDown.bCamInExecute:=TRUE;		
	
//负到正_缓存轴凸轮耦合
	fbCamInGMBuffer.iTableSel:=2;
	fbCamInGMBuffer.bCamInExecute:=TRUE;					
//负到正_隔膜平移轴凸轮耦合
	fbCamInGMDanserMove.iTableSel:=2;
	fbCamInGMDanserMove.bCamInExecute:=TRUE;

	
//负到正_放卷虚轴凸轮耦合		
	fbCamInVirGMDriver.iTableSel:=2;
	fbCamInVirGMDriver.bCamInExecute:=TRUE;		
//负到正_正极搬运平移轴凸轮耦合	
	fbAnCamInCarryingLine.ParCamIn.SlaveScaling:=-1;
	fbAnCamInCarryingLine.bCamInExecute:=TRUE;															
//负到正_正极搬运升降轴取片凸轮耦合
	fbAnCamInCarryingUpDown.iTableSel:=3;    //20240528SJ
	fbAnCamInCarryingUpDown.bCamInExecute:=TRUE;
//负到正_正极叠片平移轴凸轮耦合
	fbAnCamInDTCarryingLine.ParCamIn.SlaveScaling:=-1;
	fbAnCamInDTCarryingLine.bCamInExecute:=TRUE;	

//负到正_正极叠片升降轴取片凸轮耦合
	fbAnCamInDTCarryingUpDown.iTableSel:=3;//20240528SJ
	fbAnCamInDTCarryingUpDown.bCamInExecute:=TRUE;
//负到正_正极搬运旋转轴凸轮耦合
	fbAnCamInCarryingWhirling.ParCamIn.SlaveScaling:=-1;
	fbAnCamInCarryingWhirling.bCamInExecute:=TRUE;
//叠台左压刀升降凸轮耦合
	//fbCamInLeftYDUpDown.bCamInExecute:=TRUE;
//叠台左压刀开合凸轮耦合
	//fbCamInLeftYDLine.bCamInExecute:=TRUE;	
IF arrAxisCtrl[AxiseNo.AxisName.LeftYDLine].Cmd.arrbRealPoint[1] THEN
	fbCamInLeftYDUpDown.iTableSel:=1;
	fbCamInLeftYDLine.iTableSel:=1;
	fbCamInLeftYDUpDown.bCamInExecute:=TRUE;
	fbCamInLeftYDLine.bCamInExecute:=TRUE;	
ELSIF arrAxisCtrl[AxiseNo.AxisName.LeftYDLine].Cmd.arrbRealPoint[2] THEN	
	fbCamInLeftYDUpDown.iTableSel:=2;
	fbCamInLeftYDLine.iTableSel:=2;
	fbCamInLeftYDUpDown.bCamInExecute:=TRUE;
	fbCamInLeftYDLine.bCamInExecute:=TRUE;		
END_IF
//判断凸轮是否耦合完成
	IF fbCaCamInCarryingLine2.bInSync AND fbCaCamInDTCarryingLine.bInSync AND 
		fbCaCamInDTCarryingUpDown.bInSync  AND fbCamInGMBuffer.bInSync AND fbCamInGMDanserMove.bInSync AND
		 fbCamInVirGMDriver.bInSync AND fbAnCamInCarryingLine.bInSync AND 
		 fbCaCamInCarryingUpDown2.bInSync AND fbAnCamInCarryingUpDown.bInSync AND fbAnCamInDTCarryingUpDown.bInSync  AND 
		fbAnCamInDTCarryingLine.bInSync AND fbAnCamInCarryingWhirling.bInSync AND fbCamInLeftYDUpDown.bInSync AND
		 fbCamInLeftYDLine.bInSync  THEN
		Ca_CanIn5:=FALSE;
		//DP_Step0:=161;
	END_IF		
END_IF		

//
IF Ca_CanIn6 THEN   //OK
//负到正_负极搬运平移2轴凸轮耦合
	fbCaCamInCarryingLine2.ParCamIn.SlaveScaling:=1;
	fbCaCamInCarryingLine2.bCamInExecute:=TRUE;
//负到正_负极搬运升降2轴放片凸轮耦合
	fbCaCamInCarryingUpDown2.iTableSel:=3;  //20240528SJ
	fbCaCamInCarryingUpDown2.bCamInExecute:=TRUE;
//负到正_负极叠片平移轴凸轮耦合
	fbCaCamInDTCarryingLine.ParCamIn.SlaveScaling:=1;
	fbCaCamInDTCarryingLine.bCamInExecute:=TRUE;
//负到正_负极叠片升降轴放片凸轮耦合
	
		fbCaCamInDTCarryingUpDown.iTableSel:=2;
		fbCaCamInDTCarryingUpDown.bCamInExecute:=TRUE;
	
//叠台左压刀升降凸轮耦合
	//fbCamInLeftYDUpDown.bCamInExecute:=TRUE;
//叠台左压刀开合凸轮耦合
	//fbCamInLeftYDLine.bCamInExecute:=TRUE;	
IF arrAxisCtrl[AxiseNo.AxisName.LeftYDLine].Cmd.arrbRealPoint[1] THEN
	fbCamInLeftYDUpDown.iTableSel:=1;
	fbCamInLeftYDLine.iTableSel:=1;
	fbCamInLeftYDUpDown.bCamInExecute:=TRUE;
	fbCamInLeftYDLine.bCamInExecute:=TRUE;	
ELSIF arrAxisCtrl[AxiseNo.AxisName.LeftYDLine].Cmd.arrbRealPoint[2] THEN	
	fbCamInLeftYDUpDown.iTableSel:=2;
	fbCamInLeftYDLine.iTableSel:=2;
	fbCamInLeftYDUpDown.bCamInExecute:=TRUE;
	fbCamInLeftYDLine.bCamInExecute:=TRUE;		
END_IF
//判断凸轮耦合是否完成
	IF 	fbCaCamInCarryingLine2.bInSync AND fbCaCamInDTCarryingLine.bInSync AND 	fbCaCamInDTCarryingUpDown.bInSync  AND fbCaCamInCarryingUpDown2.bInSync AND  
		fbCamInLeftYDUpDown.bInSync AND fbCamInLeftYDLine.bInSync 	 THEN
		Ca_CanIn6:=FALSE;
		//DP_Step0:=141;
	END_IF	
END_IF		



//
IF Ca_CanIn7 THEN   //OK
//负到正_负极搬运平移2轴凸轮耦合
	fbCaCamInCarryingLine2.ParCamIn.SlaveScaling:=1;
	fbCaCamInCarryingLine2.bCamInExecute:=TRUE;						
//负到正_负极搬运升降2轴放片凸轮耦合
	fbCaCamInCarryingUpDown2.iTableSel:=3;  //20240528SJ   
	fbCaCamInCarryingUpDown2.bCamInExecute:=TRUE;
//负到正_负极叠片平移轴凸轮耦合
	fbCaCamInDTCarryingLine.ParCamIn.SlaveScaling:=1;
	fbCaCamInDTCarryingLine.bCamInExecute:=TRUE;						
//负到正_负极叠片升降轴放片凸轮耦合
		fbCaCamInDTCarryingUpDown.iTableSel:=2;
		fbCaCamInDTCarryingUpDown.bCamInExecute:=TRUE;
	
//负到正_缓存轴凸轮耦合	
	fbCamInGMBuffer.iTableSel:=2;
	fbCamInGMBuffer.bCamInExecute:=TRUE;
//负到正_隔膜平移轴凸轮耦合
	fbCamInGMDanserMove.iTableSel:=2;
	fbCamInGMDanserMove.bCamInExecute:=TRUE;

//负到正_放卷虚轴凸轮耦合
	fbCamInVirGMDriver.iTableSel:=2;
	fbCamInVirGMDriver.bCamInExecute:=TRUE;
//叠台左压刀升降凸轮耦合
	//fbCamInLeftYDUpDown.bCamInExecute:=TRUE;
//叠台左压刀开合凸轮耦合
	//fbCamInLeftYDLine.bCamInExecute:=TRUE;	
IF arrAxisCtrl[AxiseNo.AxisName.LeftYDLine].Cmd.arrbRealPoint[1] THEN
	fbCamInLeftYDUpDown.iTableSel:=1;
	fbCamInLeftYDLine.iTableSel:=1;
	fbCamInLeftYDUpDown.bCamInExecute:=TRUE;
	fbCamInLeftYDLine.bCamInExecute:=TRUE;	
ELSIF arrAxisCtrl[AxiseNo.AxisName.LeftYDLine].Cmd.arrbRealPoint[2] THEN	
	fbCamInLeftYDUpDown.iTableSel:=2;
	fbCamInLeftYDLine.iTableSel:=2;
	fbCamInLeftYDUpDown.bCamInExecute:=TRUE;
	fbCamInLeftYDLine.bCamInExecute:=TRUE;		
END_IF			
//判断凸轮耦合是否完成
	IF fbCaCamInCarryingLine2.bInSync AND fbCaCamInDTCarryingLine.bInSync AND fbCaCamInCarryingUpDown2.bInSync AND 
		fbCaCamInDTCarryingUpDown.bInSync  AND fbCamInGMBuffer.bInSync AND fbCamInGMDanserMove.bInSync AND 
		fbCamInVirGMDriver.bInSync AND fbCamInLeftYDUpDown.bInSync AND fbCamInLeftYDLine.bInSync    THEN								
			Ca_CanIn7:=FALSE;
		//DP_Step0:=141;
	END_IF
END_IF
//
IF Ca_CanIn8 THEN   //OK
//负到正_负极搬运平移2轴凸轮耦合
	fbCaCamInCarryingLine2.ParCamIn.SlaveScaling:=1;
	fbCaCamInCarryingLine2.bCamInExecute:=TRUE;
//负到正_负极搬运升降2轴放片凸轮耦合
	fbCaCamInCarryingUpDown2.iTableSel:=2;
	fbCaCamInCarryingUpDown2.bCamInExecute:=TRUE;
//负到正_负极叠片平移轴凸轮耦合
	fbCaCamInDTCarryingLine.ParCamIn.SlaveScaling:=1;
	fbCaCamInDTCarryingLine.bCamInExecute:=TRUE;
//负到正_负极叠片升降轴放片凸轮耦合
	fbCaCamInDTCarryingUpDown.iTableSel:=3;   //20240528SJ
	fbCaCamInDTCarryingUpDown.bCamInExecute:=TRUE;
//叠台左压刀升降凸轮耦合
	//fbCamInLeftYDUpDown.bCamInExecute:=TRUE;
//叠台左压刀开合凸轮耦合
	//fbCamInLeftYDLine.bCamInExecute:=TRUE;	
//判断凸轮耦合是否完成
	IF 	fbCaCamInCarryingLine2.bInSync AND fbCaCamInCarryingUpDown2	.bInSync AND 	fbCaCamInDTCarryingLine.bInSync AND fbCaCamInDTCarryingUpDown.bInSync        (*AND 	fbCaCamInDTCarryingUpDown.bInSync AND 
		fbCamInLeftYDUpDown.bInSync AND fbCamInLeftYDLine.bInSync*) 	 THEN
		Ca_CanIn8:=FALSE;
		//DP_Step0:=141;
	END_IF	
END_IF





//
IF An_CanIn1 THEN   //OK
//正到负_正极送片搬运平 移轴凸轮耦合
	fbAnCamInCarryingLine.ParCamIn.SlaveScaling:=1;
	fbAnCamInCarryingLine.bCamInExecute:=TRUE;
//正到负_正极送片搬运升降轴放片凸轮耦合
	fbAnCamInCarryingUpDown.iTableSel:=2;
	fbAnCamInCarryingUpDown.bCamInExecute:=TRUE;
//正到负_正极叠片平移轴凸轮耦合
	fbAnCamInDTCarryingLine.ParCamIn.SlaveScaling:=1;
	fbAnCamInDTCarryingLine.bCamInExecute:=TRUE;
//正到负_正极叠片升降轴放片凸轮耦合
	fbAnCamInDTCarryingUpDown.iTableSel:=2;
	fbAnCamInDTCarryingUpDown.bCamInExecute:=TRUE;
//正到负_正极搬运旋转轴凸轮耦合
fbAnCamInCarryingWhirling.ParCamIn.SlaveScaling:=1;
fbAnCamInCarryingWhirling.bCamInExecute:=TRUE;
//正到负_ 缓存轴轮耦合
	fbCamInGMBuffer.iTableSel:=1;
	 fbCamInGMBuffer.bCamInExecute:=TRUE;
//正到负_隔膜平移轴凸轮耦合
	fbCamInGMDanserMove.iTableSel:=1;
	fbCamInGMDanserMove.bCamInExecute:=TRUE;

	
//正到负_放卷虚轴凸轮耦合
	 fbCamInVirGMDriver.iTableSel :=1;
	 fbCamInVirGMDriver.bCamInExecute:=TRUE;						
//正到负_右压刀升降凸轮耦合
	//fbCamInRightYDUpDown.bCamInExecute:=TRUE;
//正极负_右压刀开合凸轮耦合
	//fbCamInRightYDLine.bCamInExecute:=TRUE;
IF arrAxisCtrl[AxiseNo.AxisName.RightYDLine].Cmd.arrbRealPoint[1] THEN	
	fbCamInRightYDUpDown.iTableSel:=1;
	fbCamInRightYDLine.iTableSel:=1;
	fbCamInRightYDUpDown.bCamInExecute:=TRUE;
    fbCamInRightYDLine.bCamInExecute:=TRUE;
ELSIF arrAxisCtrl[AxiseNo.AxisName.RightYDLine].Cmd.arrbRealPoint[2] THEN		
	fbCamInRightYDUpDown.iTableSel:=2;
	fbCamInRightYDLine.iTableSel:=2;
	fbCamInRightYDUpDown.bCamInExecute:=TRUE;
    fbCamInRightYDLine.bCamInExecute:=TRUE;	
END_IF	
//I判断凸轮耦合是否完成
	IF fbAnCamInCarryingLine.bInSync AND fbAnCamInCarryingUpDown.bInSync AND fbAnCamInDTCarryingLine.bInSync AND
		fbAnCamInDTCarryingUpDown.bInSync AND fbAnCamInCarryingWhirling.bInSync AND fbCamInGMBuffer.bInSync AND
		fbCamInGMDanserMove.bInSync AND fbCamInVirGMDriver.bInSync  AND fbCamInRightYDUpDown.bInSync AND 
		fbCamInRightYDLine.bInSync THEN
		An_CanIn1:=FALSE;
		//DP_Step0:=541;															
	END_IF					
END_IF
//
IF An_CanIn2 THEN  //OK
//正到负_正极送片搬运平移轴凸轮耦合
	fbAnCamInCarryingLine.ParCamIn.SlaveScaling:=1;
	fbAnCamInCarryingLine.bCamInExecute:=TRUE;						
//正到负_正极送片搬运升降轴放片凸轮耦合
	fbAnCamInCarryingUpDown.iTableSel:=2;
	fbAnCamInCarryingUpDown.bCamInExecute:=TRUE;
//正到负_正极叠片平移轴凸轮耦合
	fbAnCamInDTCarryingLine.ParCamIn.SlaveScaling:=1;
	fbAnCamInDTCarryingLine.bCamInExecute:=TRUE;					
//正到负_正极叠片升降轴放片凸轮耦合
	fbAnCamInDTCarryingUpDown.iTableSel:=2;
	fbAnCamInDTCarryingUpDown.bCamInExecute:=TRUE;
//正到负_正极搬运旋转轴凸轮耦合		
	fbAnCamInCarryingWhirling.ParCamIn.SlaveScaling:=1;
	fbAnCamInCarryingWhirling.bCamInExecute:=TRUE;			
//正到负_右压刀升降凸轮耦合
	//fbCamInRightYDUpDown.bCamInExecute:=TRUE;
//正极负_右压刀开合凸轮耦合
	//fbCamInRightYDLine.bCamInExecute:=TRUE;	
IF arrAxisCtrl[AxiseNo.AxisName.RightYDLine].Cmd.arrbRealPoint[1] THEN	
	fbCamInRightYDUpDown.iTableSel:=1;
	fbCamInRightYDLine.iTableSel:=1;
	fbCamInRightYDUpDown.bCamInExecute:=TRUE;
    fbCamInRightYDLine.bCamInExecute:=TRUE;
ELSIF arrAxisCtrl[AxiseNo.AxisName.RightYDLine].Cmd.arrbRealPoint[2] THEN		
	fbCamInRightYDUpDown.iTableSel:=2;
	fbCamInRightYDLine.iTableSel:=2;
	fbCamInRightYDUpDown.bCamInExecute:=TRUE;
    fbCamInRightYDLine.bCamInExecute:=TRUE;	
END_IF						 
//判断凸轮耦合是否完成
	IF fbAnCamInCarryingLine.bInSync AND fbAnCamInCarryingUpDown.bInSync AND fbAnCamInDTCarryingLine.bInSync AND fbAnCamInDTCarryingUpDown.bInSync AND 
		fbAnCamInCarryingWhirling.bInSync AND fbCamInRightYDUpDown.bInSync AND fbCamInRightYDLine.bInSync THEN
		An_CanIn2:=FALSE;
		//DP_Step0:=541;						
	END_IF			
END_IF

//
IF An_CanIn3 THEN    //OK
//正到负_正极送片搬运平移轴凸轮耦合
	fbAnCamInCarryingLine.ParCamIn.SlaveScaling:=1;
	fbAnCamInCarryingLine.bCamInExecute:=TRUE;	
//正到负_正极送片搬运升降轴放片凸轮耦合
	fbAnCamInCarryingUpDown.iTableSel:=2;
	fbAnCamInCarryingUpDown.bCamInExecute:=TRUE;
//正到负_正极叠片平移轴凸轮耦合
	fbAnCamInDTCarryingLine.ParCamIn.SlaveScaling:=1;
	fbAnCamInDTCarryingLine.bCamInExecute:=TRUE;	
//正到负_正极叠片升降轴放片凸轮耦合
	fbAnCamInDTCarryingUpDown.iTableSel:=2;
	fbAnCamInDTCarryingUpDown.bCamInExecute:=TRUE;
//正到负_正极搬运旋转轴凸轮耦合		
	fbAnCamInCarryingWhirling.ParCamIn.SlaveScaling:=1;
	fbAnCamInCarryingWhirling.bCamInExecute:=TRUE;		
//正到负_负极送片搬运平移轴凸轮耦合
	fbCaCamInCarryingLine2.ParCamIn.SlaveScaling:=-1;
	fbCaCamInCarryingLine2.bCamInExecute:=TRUE;
	
//正到负_负极送片搬运升降轴取片凸轮耦合 
  IF Mach_Control.U.EmptyRunMode THEN
	 fbCaCamInCarryingUpDown2.iTableSel:=3;
	 fbCaCamInCarryingUpDown2.bCamInExecute:=TRUE;//20240509 CF    //20240528SJ   NOT Mach_Control.U.EmptyRunMode
  ELSE
	 fbCaCamInCarryingUpDown2.iTableSel:=1;
	 fbCaCamInCarryingUpDown2.bCamInExecute:=TRUE;//20240509 CF    //20240528SJ   NOT Mach_Control.U.EmptyRunMode	  
  END_IF
	 
	 
//正到负_负极叠片搬运平移轴凸轮耦合
	fbCaCamInDTCarryingLine.ParCamIn.SlaveScaling:=-1;
	fbCaCamInDTCarryingLine.bCamInExecute:=TRUE;
//正到负_负极叠片搬运升降轴取片凸轮耦合
	fbCaCamInDTCarryingUpDown.iTableSel:=1;
	fbCaCamInDTCarryingUpDown.bCamInExecute:=TRUE;
//正到负_负极叠片搬运升降轴取片凸轮耦合
	IF iCaCamInSel2=1 THEN
		fbCaCamInDTCarryingUpDown.iTableSel:=1;
		fbCaCamInDTCarryingUpDown.bCamInExecute:=TRUE;
	END_IF	
//正到负_ 缓存轴轮耦合
	fbCamInGMBuffer.iTableSel:=1;
	 fbCamInGMBuffer.bCamInExecute:=TRUE;
//正到负_隔膜平移轴凸轮耦合
	fbCamInGMDanserMove.iTableSel:=1;
	fbCamInGMDanserMove.bCamInExecute:=TRUE;
	


//正到负_放卷虚轴凸轮耦合
	 fbCamInVirGMDriver.iTableSel :=1;
	 fbCamInVirGMDriver.bCamInExecute:=TRUE;									
//正到负_右压刀升降凸轮耦合
	//fbCamInRightYDUpDown.bCamInExecute:=TRUE;
//正极负_右压刀开合凸轮耦合
	//fbCamInRightYDLine.bCamInExecute:=TRUE;	
IF arrAxisCtrl[AxiseNo.AxisName.RightYDLine].Cmd.arrbRealPoint[1] THEN	
	fbCamInRightYDUpDown.iTableSel:=1;
	fbCamInRightYDLine.iTableSel:=1;
	fbCamInRightYDUpDown.bCamInExecute:=TRUE;
    fbCamInRightYDLine.bCamInExecute:=TRUE;
ELSIF arrAxisCtrl[AxiseNo.AxisName.RightYDLine].Cmd.arrbRealPoint[2] THEN		
	fbCamInRightYDUpDown.iTableSel:=2;
	fbCamInRightYDLine.iTableSel:=2;
	fbCamInRightYDUpDown.bCamInExecute:=TRUE;
    fbCamInRightYDLine.bCamInExecute:=TRUE;	
END_IF		
//判断凸轮是否耦合完成
	IF fbAnCamInCarryingLine.bInSync AND fbAnCamInCarryingUpDown.bInSync AND fbAnCamInDTCarryingLine.bInSync AND fbAnCamInDTCarryingUpDown.bInSync AND 
		fbAnCamInCarryingWhirling.bInSync AND fbCaCamInCarryingLine2.bInSync AND (fbCaCamInCarryingUpDown2.bInSync OR  Mach_Control.U.EmptyRunMode)
		AND fbCaCamInDTCarryingLine.bInSync AND 
		fbCaCamInDTCarryingUpDown.bInSync AND fbCamInGMBuffer.bInSync AND fbCamInGMDanserMove.bInSync AND fbCamInVirGMDriver.bInSync   AND
		fbCamInRightYDUpDown.bInSync AND fbCamInRightYDLine.bInSync  AND
		( ( fbCaCamInDTCarryingUpDown.bInSync AND iCaCamInSel2=1 ) OR   iCaCamInSel2=2 )       THEN
		An_CanIn3:=FALSE;
		//DP_Step0:=561;
	END_IF
END_IF
//

IF An_CanIn4 THEN    //OK
//正到负_正极送片搬运平移轴凸轮耦合
	fbAnCamInCarryingLine.ParCamIn.SlaveScaling:=1;
	fbAnCamInCarryingLine.bCamInExecute:=TRUE;	
//正到负_正极送片搬运升降轴放片凸轮耦合
	fbAnCamInCarryingUpDown.iTableSel:=2;
	fbAnCamInCarryingUpDown.bCamInExecute:=TRUE;
//正到负_正极叠片平移轴凸轮耦合
	fbAnCamInDTCarryingLine.ParCamIn.SlaveScaling:=1;
	fbAnCamInDTCarryingLine.bCamInExecute:=TRUE;	
//正到负_正极叠片升降轴放片凸轮耦合
	fbAnCamInDTCarryingUpDown.iTableSel:=2;
	fbAnCamInDTCarryingUpDown.bCamInExecute:=TRUE;
//正到负_正极搬运旋转轴凸轮耦合		
	fbAnCamInCarryingWhirling.ParCamIn.SlaveScaling:=1;
	fbAnCamInCarryingWhirling.bCamInExecute:=TRUE;		
//正到负_负极送片搬运平移轴凸轮耦合
	fbCaCamInCarryingLine2.ParCamIn.SlaveScaling:=-1;
	fbCaCamInCarryingLine2.bCamInExecute:=TRUE;
//正到负_负极送片搬运升降轴取片凸轮耦合 
	fbCaCamInCarryingUpDown2.iTableSel:=3; //20240528SJ
	 fbCaCamInCarryingUpDown2.bCamInExecute:=TRUE;
//正到负_负极叠片搬运平移轴凸轮耦合
	fbCaCamInDTCarryingLine.ParCamIn.SlaveScaling:=-1;
	fbCaCamInDTCarryingLine.bCamInExecute:=TRUE;
//正到负_负极叠片搬运升降轴取片凸轮耦合
	fbCaCamInDTCarryingUpDown.iTableSel:=1;
	fbCaCamInDTCarryingUpDown.bCamInExecute:=TRUE;						
//正到负_右压刀升降凸轮耦合
	//fbCamInRightYDUpDown.bCamInExecute:=TRUE;
//正极负_右压刀开合凸轮耦合
	//fbCamInRightYDLine.bCamInExecute:=TRUE;	
IF arrAxisCtrl[AxiseNo.AxisName.RightYDLine].Cmd.arrbRealPoint[1] THEN	
	fbCamInRightYDUpDown.iTableSel:=1;
	fbCamInRightYDLine.iTableSel:=1;
	fbCamInRightYDUpDown.bCamInExecute:=TRUE;
    fbCamInRightYDLine.bCamInExecute:=TRUE;
ELSIF arrAxisCtrl[AxiseNo.AxisName.RightYDLine].Cmd.arrbRealPoint[2] THEN		
	fbCamInRightYDUpDown.iTableSel:=2;
	fbCamInRightYDLine.iTableSel:=2;
	fbCamInRightYDUpDown.bCamInExecute:=TRUE;
    fbCamInRightYDLine.bCamInExecute:=TRUE;	
END_IF		
//判断凸轮是否耦合完成
	IF fbAnCamInCarryingLine.bInSync AND fbAnCamInCarryingUpDown.bInSync AND fbAnCamInDTCarryingLine.bInSync AND fbAnCamInDTCarryingUpDown.bInSync AND 
		fbAnCamInCarryingWhirling.bInSync AND fbCaCamInCarryingLine2.bInSync AND fbCaCamInCarryingUpDown2.bInSync   AND fbCaCamInDTCarryingLine.bInSync AND 
		fbCaCamInDTCarryingUpDown.bInSync AND fbCamInRightYDUpDown.bInSync AND fbCamInRightYDLine.bInSync THEN
		An_CanIn4:=FALSE;
		//DP_Step0:=561;								
	END_IF
END_IF


//
IF An_CanIn5 THEN     //OK
//正到负_正极送片搬运平移轴凸轮耦合
	fbAnCamInCarryingLine.ParCamIn.SlaveScaling:=1;
	fbAnCamInCarryingLine.bCamInExecute:=TRUE;	
//正到负_正极送片搬运升降轴放片凸轮耦合
	fbAnCamInCarryingUpDown.iTableSel:=3;  //20240528SJ
	fbAnCamInCarryingUpDown.bCamInExecute:=TRUE;
//正到负_正极叠片平移轴凸轮耦合
	fbAnCamInDTCarryingLine.ParCamIn.SlaveScaling:=1;
	fbAnCamInDTCarryingLine.bCamInExecute:=TRUE;	
//正到负_正极叠片升降轴放片凸轮耦合
	//IF NOT KD_Mark THEN//空叠隔膜中
		fbAnCamInDTCarryingUpDown.iTableSel:=2;
		fbAnCamInDTCarryingUpDown.bCamInExecute:=TRUE;
	//END_IF
//正到负_正极搬运旋转轴凸轮耦合		
	fbAnCamInCarryingWhirling.ParCamIn.SlaveScaling:=1;
	fbAnCamInCarryingWhirling.bCamInExecute:=TRUE;		
//正到负_负极送片搬运平移轴凸轮耦合
	fbCaCamInCarryingLine2.ParCamIn.SlaveScaling:=-1;
	fbCaCamInCarryingLine2.bCamInExecute:=TRUE;
//正到负_负极送片搬运升降轴取片凸轮耦合 
	 fbCaCamInCarryingUpDown2.iTableSel:=3;   //20240528SJ
	fbCaCamInCarryingUpDown2.bCamInExecute:=TRUE;
//正到负_负极叠片搬运平移轴凸轮耦合
	fbCaCamInDTCarryingLine.ParCamIn.SlaveScaling:=-1;
	fbCaCamInDTCarryingLine.bCamInExecute:=TRUE;
//正到负_负极叠片搬运升降轴取片凸轮耦合
	fbCaCamInDTCarryingUpDown.iTableSel:=3;   //20240528SJ
	fbCaCamInDTCarryingUpDown.bCamInExecute:=TRUE;
//正到负_ 缓存轴轮耦合
	 fbCamInGMBuffer.iTableSel:=1;
	 fbCamInGMBuffer.bCamInExecute:=TRUE;
//正到负_隔膜平移轴凸轮耦合
	fbCamInGMDanserMove.iTableSel:=1;
	fbCamInGMDanserMove.bCamInExecute:=TRUE;
	
				
//正到负_放卷虚轴凸轮耦合
	 fbCamInVirGMDriver.iTableSel :=1;
	 fbCamInVirGMDriver.bCamInExecute:=TRUE;									
//正到负_右压刀升降凸轮耦合
	//fbCamInRightYDUpDown.bCamInExecute:=TRUE;
//正极负_右压刀开合凸轮耦合
	//fbCamInRightYDLine.bCamInExecute:=TRUE;	
IF arrAxisCtrl[AxiseNo.AxisName.RightYDLine].Cmd.arrbRealPoint[1] THEN	
	fbCamInRightYDUpDown.iTableSel:=1;
	fbCamInRightYDLine.iTableSel:=1;
	fbCamInRightYDUpDown.bCamInExecute:=TRUE;
    fbCamInRightYDLine.bCamInExecute:=TRUE;
ELSIF arrAxisCtrl[AxiseNo.AxisName.RightYDLine].Cmd.arrbRealPoint[2] THEN		
	fbCamInRightYDUpDown.iTableSel:=2;
	fbCamInRightYDLine.iTableSel:=2;
	fbCamInRightYDUpDown.bCamInExecute:=TRUE;
    fbCamInRightYDLine.bCamInExecute:=TRUE;	
END_IF		
//判断凸轮是否耦合完成
	IF fbAnCamInCarryingLine.bInSync AND fbAnCamInDTCarryingLine.bInSync AND fbAnCamInDTCarryingUpDown.bInSync AND 
		fbAnCamInCarryingWhirling.bInSync AND fbCaCamInCarryingLine2.bInSync AND 
		fbAnCamInCarryingUpDown.bInSync AND  fbCaCamInCarryingUpDown2.bInSync AND fbCaCamInDTCarryingUpDown.bInSync  AND  //20240528SJ
		fbCamInGMBuffer.bInSync AND fbCamInGMDanserMove.bInSync AND fbCamInVirGMDriver.bInSync   AND
		fbCamInRightYDUpDown.bInSync AND fbCamInRightYDLine.bInSync         THEN
		An_CanIn5:=FALSE;
		//DP_Step0:=561;
	END_IF
END_IF				

IF An_CanIn6 THEN   //OK
//正到负_正极送片搬运平 移轴凸轮耦合
	fbAnCamInCarryingLine.ParCamIn.SlaveScaling:=1;
	fbAnCamInCarryingLine.bCamInExecute:=TRUE;
//正到负_正极送片搬运升降轴放片凸轮耦合
	fbAnCamInCarryingUpDown.iTableSel:=3;   //20240528SJ
	fbAnCamInCarryingUpDown.bCamInExecute:=TRUE;
//正到负_正极叠片平移轴凸轮耦合
	fbAnCamInDTCarryingLine.ParCamIn.SlaveScaling:=1;
	fbAnCamInDTCarryingLine.bCamInExecute:=TRUE;
//正到负_正极叠片升降轴放片凸轮耦合
	//IF NOT KD_Mark THEN//空叠隔膜中
		fbAnCamInDTCarryingUpDown.iTableSel:=2;
		fbAnCamInDTCarryingUpDown.bCamInExecute:=TRUE;
	//END_IF
//正到负_正极搬运旋转轴凸轮耦合
fbAnCamInCarryingWhirling.ParCamIn.SlaveScaling:=1;
fbAnCamInCarryingWhirling.bCamInExecute:=TRUE;
//正到负_ 缓存轴轮耦合
	fbCamInGMBuffer.iTableSel:=1;
	 fbCamInGMBuffer.bCamInExecute:=TRUE;
//正到负_隔膜平移轴凸轮耦合
	fbCamInGMDanserMove.iTableSel:=1;
	fbCamInGMDanserMove.bCamInExecute:=TRUE;

	
//正到负_放卷虚轴凸轮耦合
	 fbCamInVirGMDriver.iTableSel :=1;
	 fbCamInVirGMDriver.bCamInExecute:=TRUE;						
//正到负_右压刀升降凸轮耦合
	//fbCamInRightYDUpDown.bCamInExecute:=TRUE;
//正极负_右压刀开合凸轮耦合
	//fbCamInRightYDLine.bCamInExecute:=TRUE;
IF arrAxisCtrl[AxiseNo.AxisName.RightYDLine].Cmd.arrbRealPoint[1] THEN	
	fbCamInRightYDUpDown.iTableSel:=1;
	fbCamInRightYDLine.iTableSel:=1;
	fbCamInRightYDUpDown.bCamInExecute:=TRUE;
    fbCamInRightYDLine.bCamInExecute:=TRUE;
ELSIF arrAxisCtrl[AxiseNo.AxisName.RightYDLine].Cmd.arrbRealPoint[2] THEN		
	fbCamInRightYDUpDown.iTableSel:=2;
	fbCamInRightYDLine.iTableSel:=2;
	fbCamInRightYDUpDown.bCamInExecute:=TRUE;
    fbCamInRightYDLine.bCamInExecute:=TRUE;	
END_IF		
//I判断凸轮耦合是否完成
	IF fbAnCamInCarryingLine.bInSync AND  fbAnCamInDTCarryingLine.bInSync AND  fbAnCamInCarryingUpDown.bInSync AND 
		fbAnCamInDTCarryingUpDown.bInSync AND fbAnCamInCarryingWhirling.bInSync AND fbCamInGMBuffer.bInSync AND
		fbCamInGMDanserMove.bInSync AND fbCamInVirGMDriver.bInSync  AND fbCamInRightYDUpDown.bInSync AND 
		fbCamInRightYDLine.bInSync THEN
		An_CanIn6:=FALSE;
		//DP_Step0:=541;															
	END_IF					
END_IF				


//
IF An_CanIn7 THEN  //OK
//正到负_正极送片搬运平移轴凸轮耦合
	fbAnCamInCarryingLine.ParCamIn.SlaveScaling:=1;
	fbAnCamInCarryingLine.bCamInExecute:=TRUE;						
//正到负_正极送片搬运升降轴放片凸轮耦合
	fbAnCamInCarryingUpDown.iTableSel:=3;  //20240528SJ
	fbAnCamInCarryingUpDown.bCamInExecute:=TRUE;
//正到负_正极叠片平移轴凸轮耦合
	fbAnCamInDTCarryingLine.ParCamIn.SlaveScaling:=1;
	fbAnCamInDTCarryingLine.bCamInExecute:=TRUE;					
//正到负_正极叠片升降轴放片凸轮耦合
	
		fbAnCamInDTCarryingUpDown.iTableSel:=2;
		fbAnCamInDTCarryingUpDown.bCamInExecute:=TRUE;
	
//正到负_正极搬运旋转轴凸轮耦合		
	fbAnCamInCarryingWhirling.ParCamIn.SlaveScaling:=1;
	fbAnCamInCarryingWhirling.bCamInExecute:=TRUE;			
//正到负_右压刀升降凸轮耦合
	//fbCamInRightYDUpDown.bCamInExecute:=TRUE;
//正极负_右压刀开合凸轮耦合
	//fbCamInRightYDLine.bCamInExecute:=TRUE;	
IF arrAxisCtrl[AxiseNo.AxisName.RightYDLine].Cmd.arrbRealPoint[1] THEN	
	fbCamInRightYDUpDown.iTableSel:=1;
	fbCamInRightYDLine.iTableSel:=1;
	fbCamInRightYDUpDown.bCamInExecute:=TRUE;
    fbCamInRightYDLine.bCamInExecute:=TRUE;
ELSIF arrAxisCtrl[AxiseNo.AxisName.RightYDLine].Cmd.arrbRealPoint[2] THEN		
	fbCamInRightYDUpDown.iTableSel:=2;
	fbCamInRightYDLine.iTableSel:=2;
	fbCamInRightYDUpDown.bCamInExecute:=TRUE;
    fbCamInRightYDLine.bCamInExecute:=TRUE;	
END_IF						 
//判断凸轮耦合是否完成
	IF fbAnCamInCarryingLine.bInSync AND  fbAnCamInDTCarryingLine.bInSync AND fbAnCamInDTCarryingUpDown.bInSync  AND    fbAnCamInCarryingUpDown.bInSync AND 
		fbAnCamInCarryingWhirling.bInSync AND fbCamInRightYDUpDown.bInSync AND fbCamInRightYDLine.bInSync THEN
		An_CanIn7:=FALSE;
		//DP_Step0:=541;						
	END_IF			
END_IF
END_ACTION

ACTION _01DT_AutoSub1_CamOut:
CamOut_TON(IN:= , PT:=T#10MS , Q=> , ET=> );



//判断是否有叠台部分轴在耦合中
				IF 	NOT arrAxis[AxiseNo.AxisName.AnCarryingLine].Status.Coupled AND NOT arrAxis[AxiseNo.AxisName.AnCarryingUpDown].Status.Coupled AND 
					NOT arrAxis[AxiseNo.AxisName.AnDTCarryingLine].Status.Coupled AND NOT arrAxis[AxiseNo.AxisName.AnDTCarryingUpDown].Status.Coupled AND 
					NOT arrAxis[AxiseNo.AxisName.AnCarryingWhirling].Status.Coupled AND NOT arrAxis[AxiseNo.AxisName.CaCarryingLine2].Status.Coupled AND 
					NOT arrAxis[AxiseNo.AxisName.CaCarryingUpDown2].Status.Coupled AND NOT arrAxis[AxiseNo.AxisName.CaDTCarryingLine].Status.Coupled AND 
					NOT arrAxis[AxiseNo.AxisName.CaDTCarryingUpDown].Status.Coupled AND NOT arrAxis[AxiseNo.AxisName.LeftYDLine].Status.Coupled AND 
					NOT arrAxis[AxiseNo.AxisName.LeftYDUpDown].Status.Coupled AND NOT arrAxis[AxiseNo.AxisName.RightYDLine].Status.Coupled AND 
					NOT arrAxis[AxiseNo.AxisName.RightYDUpDown].Status.Coupled AND NOT arrAxis[AxiseNo.AxisName.SEPTATCache].Status.Coupled AND 
					NOT arrAxis[AxiseNo.AxisName.SEPTATLine].Status.Coupled AND NOT arrAxis[AxiseNo.VirAxisName.VirTailCurl].Status.Coupled 
					  THEN  //NOT arrAxis[AxiseNo.VirAxisName.VirGM].Status.Coupled
					DT_AxiseCoupling:=FALSE;//叠片部分轴在耦合中
				ELSE
					DT_AxiseCoupling:=TRUE;
				END_IF
//叠台自动子程序_凸轮耦合解除_主轴清零
rDTCamOut_TRIG(CLK:=Mach_Control.DT_b.DT_AllCamOut OR arrAxisCamError , Q=> );
IF   rDTCamOut_TRIG.Q    THEN
	DP_Step1:=100;
END_IF


IF DP_Step1=100 THEN
	            DPtime1:=1;
				CamOut_TON.IN:=FALSE;
				IF arrAxisCtrl[AxiseNo.VirAxisName.VirMain].Status.NoMoving  THEN
					arrAxisCtrl[AxiseNo.VirAxisName.VirMain].Cmd.bStop:=FALSE;
					fbAnCamInCarryingLine.bCamInExecute:=FALSE;//正极送片搬运平移
					fbAnCamInCarryingUpDown.bCamInExecute:=FALSE;//正极送片搬运升降
					fbAnCamInCarryingWhirling.bCamInExecute:=FALSE;//正极送片搬运旋转
					fbAnCamInDTCarryingLine.bCamInExecute:=FALSE;//正极叠片搬运平移
					fbAnCamInDTCarryingUpDown.bCamInExecute:=FALSE;//正极叠片搬运升降
					
					//fbCaCamInCarryingLine1.bCamInExecute,:=TURE;//负极取流水线平移
					//fbCaCamInCarryingUpDown1.bCamInExecute:=TRUE;//负极取流水线升降
					fbCaCamInCarryingLine2.bCamInExecute:=FALSE;//负极送片搬运平移
					fbCaCamInCarryingUpDown2.bCamInExecute:=FALSE;//负极送片搬运升降
					fbCaCamInDTCarryingLine.bCamInExecute:=FALSE;//负极叠片搬运平移
					fbCaCamInDTCarryingUpDown.bCamInExecute:=FALSE;//负极叠片搬运升降
					
					fbCamInLeftYDLine.bCamInExecute:=FALSE;//左压刀开合
					fbCamInLeftYDUpDown.bCamInExecute:=FALSE;//左压刀升降
					fbCamInRightYDLine.bCamInExecute:=FALSE;//右压刀开合
					fbCamInRightYDUpDown.bCamInExecute:=FALSE;//左压刀升降
					
					fbCamInGMBuffer.bCamInExecute:=FALSE;//隔膜缓存
					fbCamInGMDanserMove.bCamInExecute:=FALSE;//隔膜平移
					fbCamInVirGMDriver.bCamInExecute:=FALSE;//隔膜放卷虚轴
					
					
					fbCamInGMBuffer2.bCamInExecute:=FALSE;	//隔膜缓存2	
					fbCamInVirGMDriver2.bCamInExecute:=FALSE;	//隔膜放卷虚轴2
					
					arrAxisCtrl[AxiseNo.VirAxisName.VirMain].Cmd	.bMoveAbs:=FALSE;	
					DP_Step1:=140;
					
				ELSE
					arrAxisCtrl[AxiseNo.VirAxisName.VirMain].Cmd.bStop:=TRUE;
				END_IF
	END_IF			
	
	
IF DP_Step1=140 THEN
			IF 	NOT arrAxis[AxiseNo.AxisName.AnCarryingLine].Status.Coupled AND NOT arrAxis[AxiseNo.AxisName.AnCarryingUpDown].Status.Coupled AND 
				NOT arrAxis[AxiseNo.AxisName.AnDTCarryingLine].Status.Coupled AND NOT arrAxis[AxiseNo.AxisName.AnDTCarryingUpDown].Status.Coupled AND 
				NOT arrAxis[AxiseNo.AxisName.AnCarryingWhirling].Status.Coupled AND NOT arrAxis[AxiseNo.AxisName.CaCarryingLine2].Status.Coupled AND 
				NOT arrAxis[AxiseNo.AxisName.CaCarryingUpDown2].Status.Coupled AND NOT arrAxis[AxiseNo.AxisName.CaDTCarryingLine].Status.Coupled AND 
				NOT arrAxis[AxiseNo.AxisName.CaDTCarryingUpDown].Status.Coupled AND NOT arrAxis[AxiseNo.AxisName.LeftYDLine].Status.Coupled AND 
				NOT arrAxis[AxiseNo.AxisName.LeftYDUpDown].Status.Coupled AND NOT arrAxis[AxiseNo.AxisName.RightYDLine].Status.Coupled AND 
				NOT arrAxisCtrl[AxiseNo.AxisName.RightYDUpDown].Status.Coupled AND NOT arrAxis[AxiseNo.AxisName.SEPTATCache].Status.Coupled AND 
				NOT arrAxis[AxiseNo.AxisName.SEPTATLine].Status.Coupled   AND NOT DT_AxiseCoupling    THEN  //AND NOT arrAxis[AxiseNo.VirAxisName.VirGM].Status.Coupled
					arrAxisCtrl[AxiseNo.VirAxisName.VirMain].Cmd.fSetPos:=0;
					
					arrAxisCtrl[AxiseNo.VirAxisName.VirMain].Cmd.bSetPos:=TRUE;	
					DP_Step1:=160;
					DPtime1:=2;
			END_IF	
   END_IF
			
	IF DP_Step1=160 THEN  //判断主轴是否停止以及在模长初始位
				IF  NOT arrAxisCtrl[AxiseNo.VirAxisName.VirMain].Cmd.bSetPos AND arrAxis[AxiseNo.VirAxisName.VirMain].NcToPlc.SetPos=0   THEN
					DP_Step1:=6666;
					DPtime1:=3;
				END_IF
     END_IF






(*

CASE DP_Step1 OF
		100://先判断主轴是否在停止中
				CamOut_TON.IN:=FALSE;
				IF arrAxisCtrl[AxiseNo.VirAxisName.VirMain].Status.NoMoving  THEN
					arrAxisCtrl[AxiseNo.VirAxisName.VirMain].Cmd.bStop:=FALSE;
					fbAnCamInCarryingLine.bCamInExecute:=FALSE;//正极送片搬运平移
					fbAnCamInCarryingUpDown.bCamInExecute:=FALSE;//正极送片搬运升降
					fbAnCamInCarryingWhirling.bCamInExecute:=FALSE;//正极送片搬运旋转
					fbAnCamInDTCarryingLine.bCamInExecute:=FALSE;//正极叠片搬运平移
					fbAnCamInDTCarryingUpDown.bCamInExecute:=FALSE;//正极叠片搬运升降
					
					//fbCaCamInCarryingLine1.bCamInExecute,:=TURE;//负极取流水线平移
					//fbCaCamInCarryingUpDown1.bCamInExecute:=TRUE;//负极取流水线升降
					fbCaCamInCarryingLine2.bCamInExecute:=FALSE;//负极送片搬运平移
					fbCaCamInCarryingUpDown2.bCamInExecute:=FALSE;//负极送片搬运升降
					fbCaCamInDTCarryingLine.bCamInExecute:=FALSE;//负极叠片搬运平移
					fbCaCamInDTCarryingUpDown.bCamInExecute:=FALSE;//负极叠片搬运升降
					
					fbCamInLeftYDLine.bCamInExecute:=FALSE;//左压刀开合
					fbCamInLeftYDUpDown.bCamInExecute:=FALSE;//左压刀升降
					fbCamInRightYDLine.bCamInExecute:=FALSE;//右压刀开合
					fbCamInRightYDUpDown.bCamInExecute:=FALSE;//左压刀升降
					
					fbCamInGMBuffer.bCamInExecute:=FALSE;//隔膜缓存
					fbCamInGMDanserMove.bCamInExecute:=FALSE;//隔膜平移
					fbCamInVirGMDriver.bCamInExecute:=FALSE;//隔膜放卷虚轴
					fbCamInVirGM.bCamInExecute:=FALSE;//隔膜纠偏
					
					fbCamInGMBuffer2.bCamInExecute:=FALSE;	//隔膜缓存2	
					fbCamInVirGMDriver2.bCamInExecute:=FALSE;	//隔膜放卷虚轴2
					
					arrAxisCtrl[AxiseNo.VirAxisName.VirMain].Cmd	.bMoveAbs:=FALSE;	
					DP_Step1:=140;
				ELSE
					arrAxisCtrl[AxiseNo.VirAxisName.VirMain].Cmd.bStop:=TRUE;
				END_IF
				
		140:
			IF 	NOT arrAxisCtrl[AxiseNo.AxisName.AnCarryingLine].Status.Coupled AND NOT arrAxisCtrl[AxiseNo.AxisName.AnCarryingUpDown].Status.Coupled AND 
				NOT arrAxisCtrl[AxiseNo.AxisName.AnDTCarryingLine].Status.Coupled AND NOT arrAxisCtrl[AxiseNo.AxisName.AnDTCarryingUpDown].Status.Coupled AND 
				NOT arrAxisCtrl[AxiseNo.AxisName.AnCarryingWhirling].Status.Coupled AND NOT arrAxisCtrl[AxiseNo.AxisName.CaCarryingLine2].Status.Coupled AND 
				NOT arrAxisCtrl[AxiseNo.AxisName.CaCarryingUpDown2].Status.Coupled AND NOT arrAxisCtrl[AxiseNo.AxisName.CaDTCarryingLine].Status.Coupled AND 
				NOT arrAxisCtrl[AxiseNo.AxisName.CaDTCarryingUpDown].Status.Coupled AND NOT arrAxisCtrl[AxiseNo.AxisName.LeftYDLine].Status.Coupled AND 
				NOT arrAxisCtrl[AxiseNo.AxisName.LeftYDUpDown].Status.Coupled AND NOT arrAxisCtrl[AxiseNo.AxisName.RightYDLine].Status.Coupled AND 
				NOT arrAxisCtrl[AxiseNo.AxisName.RightYDUpDown].Status.Coupled AND NOT arrAxisCtrl[AxiseNo.AxisName.SEPTATCache].Status.Coupled AND 
				NOT arrAxisCtrl[AxiseNo.AxisName.SEPTATLine].Status.Coupled AND NOT arrAxisCtrl[AxiseNo.VirAxisName.VirGM].Status.Coupled AND NOT DT_AxiseCoupling THEN
					arrAxisCtrl[AxiseNo.VirAxisName.VirMain].Cmd.fSetPos:=0;
					arrAxisCtrl[AxiseNo.VirAxisName.VirMain].Cmd.bSetPos:=TRUE;	
					DP_Step1:=160;
			END_IF	

		160://判断主轴是否停止以及在模长初始位
				IF  NOT arrAxisCtrl[AxiseNo.VirAxisName.VirMain].Cmd.bSetPos AND arrAxis[AxiseNo.VirAxisName.VirMain].NcToPlc.SetPos=0   THEN
					DP_Step1:=6666;
				END_IF
END_CASE

(*
CamOut_TON(IN:= , PT:=T#5MS , Q=> , ET=> );



//判断是否有叠台部分轴在耦合中
				IF 	NOT arrAxisCtrl[AxiseNo.AxisName.AnCarryingLine].Status.Coupled AND NOT arrAxisCtrl[AxiseNo.AxisName.AnCarryingUpDown].Status.Coupled AND 
					NOT arrAxisCtrl[AxiseNo.AxisName.AnDTCarryingLine].Status.Coupled AND NOT arrAxisCtrl[AxiseNo.AxisName.AnDTCarryingUpDown].Status.Coupled AND 
					NOT arrAxisCtrl[AxiseNo.AxisName.AnCarryingWhirling].Status.Coupled AND NOT arrAxisCtrl[AxiseNo.AxisName.CaCarryingLine2].Status.Coupled AND 
					NOT arrAxisCtrl[AxiseNo.AxisName.CaCarryingUpDown2].Status.Coupled AND NOT arrAxisCtrl[AxiseNo.AxisName.CaDTCarryingLine].Status.Coupled AND 
					NOT arrAxisCtrl[AxiseNo.AxisName.CaDTCarryingUpDown].Status.Coupled AND NOT arrAxisCtrl[AxiseNo.AxisName.LeftYDLine].Status.Coupled AND 
					NOT arrAxisCtrl[AxiseNo.AxisName.LeftYDUpDown].Status.Coupled AND NOT arrAxisCtrl[AxiseNo.AxisName.RightYDLine].Status.Coupled AND 
					NOT arrAxisCtrl[AxiseNo.AxisName.RightYDUpDown].Status.Coupled AND NOT arrAxisCtrl[AxiseNo.AxisName.SEPTATCache].Status.Coupled AND 
					NOT arrAxisCtrl[AxiseNo.AxisName.SEPTATLine].Status.Coupled AND NOT arrAxisCtrl[AxiseNo.VirAxisName.VirTailCurl].Status.Coupled AND
					NOT arrAxisCtrl[AxiseNo.VirAxisName.VirGM].Status.Coupled  THEN
					DT_AxiseCoupling:=FALSE;//叠片部分轴在耦合中
				ELSE
					DT_AxiseCoupling:=TRUE;
				END_IF
//叠台自动子程序_凸轮耦合解除_主轴清零
rDTCamOut_TRIG(CLK:=Mach_Control.DT_b.DT_AllCamOut OR arrAxisCamError , Q=> );
IF   rDTCamOut_TRIG.Q    THEN
	DP_Step1:=100;
END_IF
CASE DP_Step1 OF
		100://先判断主轴是否在停止中
				CamOut_TON.IN:=FALSE;
				IF arrAxisCtrl[AxiseNo.VirAxisName.VirMain].Status.NoMoving  THEN
					arrAxisCtrl[AxiseNo.VirAxisName.VirMain].Cmd.bStop:=FALSE;
					DP_Step1:=120;
				ELSE
					arrAxisCtrl[AxiseNo.VirAxisName.VirMain].Cmd.bStop:=TRUE;
				END_IF
		110://判断轴是否在耦合中
				(*
						IF DT_AxiseCoupling THEN
							DP_Step1:=120;
						ELSE
							DP_Step1:=130;
						END_IF
				*)
				DP_Step1:=120;
		120://叠台部轴解除耦合
				fbAnCamInCarryingLine.bCamInExecute:=FALSE;//正极送片搬运平移
				fbAnCamInCarryingUpDown.bCamInExecute:=FALSE;//正极送片搬运升降
				fbAnCamInCarryingWhirling.bCamInExecute:=FALSE;//正极送片搬运旋转
				 fbAnCamInDTCarryingLine.bCamInExecute:=FALSE;//正极叠片搬运平移
				fbAnCamInDTCarryingUpDown.bCamInExecute:=FALSE;//正极叠片搬运升降
				
				//fbCaCamInCarryingLine1.bCamInExecute,:=TURE;//负极取流水线平移
				//fbCaCamInCarryingUpDown1.bCamInExecute:=TRUE;//负极取流水线升降
				fbCaCamInCarryingLine2.bCamInExecute:=FALSE;//负极送片搬运平移
				fbCaCamInCarryingUpDown2.bCamInExecute:=FALSE;//负极送片搬运升降
				fbCaCamInDTCarryingLine.bCamInExecute:=FALSE;//负极叠片搬运平移
				fbCaCamInDTCarryingUpDown.bCamInExecute:=FALSE;//负极叠片搬运升降
				
				fbCamInLeftYDLine.bCamInExecute:=FALSE;//左压刀开合
				fbCamInLeftYDUpDown.bCamInExecute:=FALSE;//左压刀升降
				fbCamInRightYDLine.bCamInExecute:=FALSE;//右压刀开合
				fbCamInRightYDUpDown.bCamInExecute:=FALSE;//左压刀升降
				
				fbCamInGMBuffer.bCamInExecute:=FALSE;//隔膜缓存
				fbCamInGMDanserMove.bCamInExecute:=FALSE;//隔膜平移
				fbCamInVirGMDriver.bCamInExecute:=FALSE;//隔膜放卷虚轴
				fbCamInVirGM.bCamInExecute:=FALSE;//隔膜纠偏
				IF NOT fbAnCamInCarryingLine.bCamInExecute AND NOT fbAnCamInCarryingUpDown.bCamInExecute AND 
					NOT  fbAnCamInCarryingWhirling.bCamInExecute AND NOT fbAnCamInDTCarryingLine.bCamInExecute AND 
					NOT  fbAnCamInDTCarryingUpDown.bCamInExecute AND NOT fbCaCamInCarryingLine2.bCamInExecute AND 
					NOT  fbCaCamInCarryingUpDown2.bCamInExecute AND NOT fbCaCamInDTCarryingLine.bCamInExecute AND 
					NOT  fbCaCamInDTCarryingUpDown.bCamInExecute AND NOT fbCamInLeftYDLine.bCamInExecute AND 
					NOT fbCamInLeftYDUpDown.bCamInExecute AND NOT fbCamInRightYDLine.bCamInExecute AND 
					NOT  fbCamInRightYDUpDown.bCamInExecute AND NOT fbCamInGMBuffer.bCamInExecute AND 
					NOT fbCamInGMDanserMove.bCamInExecute AND NOT fbCamInVirGMDriver.bCamInExecute AND 
					NOT fbCamInVirGM.bCamInExecute THEN
						DP_Step1:=150;
				END_IF
(*
		130:	
				arrAxisCtrl[AxiseNo.AxisName.AnCarryingLine].Cmd.bGearOut:=TRUE;
				arrAxisCtrl[AxiseNo.AxisName.AnCarryingUpDown].Cmd.bGearOut:=TRUE;
				arrAxisCtrl[AxiseNo.AxisName.AnCarryingWhirling].Cmd.bGearOut:=TRUE;
				arrAxisCtrl[AxiseNo.AxisName.AnDTCarryingLine].Cmd.bGearOut:=TRUE;
				arrAxisCtrl[AxiseNo.AxisName.AnDTCarryingUpDown].Cmd.bGearOut:=TRUE;
				arrAxisCtrl[AxiseNo.AxisName.CaCarryingLine2].Cmd.bGearOut:=TRUE;
				arrAxisCtrl[AxiseNo.AxisName.CaCarryingUpDown2].Cmd.bGearOut:=TRUE;
				arrAxisCtrl[AxiseNo.AxisName.CaDTCarryingLine].Cmd.bGearOut:=TRUE;
				arrAxisCtrl[AxiseNo.AxisName.CaDTCarryingUpDown].Cmd.bGearOut:=TRUE;
				arrAxisCtrl[AxiseNo.AxisName.LeftYDLine].Cmd.bGearOut:=TRUE;
				arrAxisCtrl[AxiseNo.AxisName.LeftYDUpDown].Cmd.bGearOut:=TRUE;
				arrAxisCtrl[AxiseNo.AxisName.RightYDLine].Cmd.bGearOut:=TRUE;
				arrAxisCtrl[AxiseNo.AxisName.RightYDUpDown].Cmd.bGearOut:=TRUE;
				arrAxisCtrl[AxiseNo.AxisName.SEPTATCache].Cmd.bGearOut:=TRUE;
				arrAxisCtrl[AxiseNo.AxisName.SEPTATLine].Cmd.bGearOut:=TRUE;
				arrAxisCtrl[AxiseNo.VirAxisName.VirGM].Cmd.bGearOut:=TRUE;
				IF NOT DT_AxiseCoupling THEN
					arrAxisCtrl[AxiseNo.AxisName.AnCarryingLine].Cmd.bGearOut:=FALSE;
					arrAxisCtrl[AxiseNo.AxisName.AnCarryingUpDown].Cmd.bGearOut:=FALSE;
					arrAxisCtrl[AxiseNo.AxisName.AnCarryingWhirling].Cmd.bGearOut:=FALSE;
					arrAxisCtrl[AxiseNo.AxisName.AnDTCarryingLine].Cmd.bGearOut:=FALSE;
					arrAxisCtrl[AxiseNo.AxisName.AnDTCarryingUpDown].Cmd.bGearOut:=FALSE;
					arrAxisCtrl[AxiseNo.AxisName.CaCarryingLine2].Cmd.bGearOut:=FALSE;
					arrAxisCtrl[AxiseNo.AxisName.CaCarryingUpDown2].Cmd.bGearOut:=FALSE;
					arrAxisCtrl[AxiseNo.AxisName.CaDTCarryingLine].Cmd.bGearOut:=FALSE;
					arrAxisCtrl[AxiseNo.AxisName.CaDTCarryingUpDown].Cmd.bGearOut:=FALSE;
					arrAxisCtrl[AxiseNo.AxisName.LeftYDLine].Cmd.bGearOut:=FALSE;
					arrAxisCtrl[AxiseNo.AxisName.LeftYDUpDown].Cmd.bGearOut:=FALSE;
					arrAxisCtrl[AxiseNo.AxisName.RightYDLine].Cmd.bGearOut:=FALSE;
					arrAxisCtrl[AxiseNo.AxisName.RightYDUpDown].Cmd.bGearOut:=FALSE;
					arrAxisCtrl[AxiseNo.AxisName.SEPTATCache].Cmd.bGearOut:=FALSE;
					arrAxisCtrl[AxiseNo.AxisName.SEPTATLine].Cmd.bGearOut:=FALSE;
					arrAxisCtrl[AxiseNo.VirAxisName.VirGM].Cmd.bGearOut:=FALSE;					
					DP_Step1:=140;
				END_IF
				
		140:
				IF NOT CamOut_TON.Q THEN
					CamOut_TON.IN:=TRUE;
				ELSE
					CamOut_TON.IN:=FALSE;
					DP_Step1:=150;
				END_IF*)
		150://主轴当前位置清零				
				arrAxisCtrl[AxiseNo.VirAxisName.VirMain].Cmd.fSetPos:=0;
				arrAxisCtrl[AxiseNo.VirAxisName.VirMain].Cmd.bSetPos:=TRUE;			
				DP_Step1:=160;

		160://判断主轴是否停止以及在模长初始位
				IF  NOT arrAxisCtrl[AxiseNo.VirAxisName.VirMain].Cmd.bSetPos AND arrAxis[AxiseNo.VirAxisName.VirMain].NcToPlc.SetPos=0   THEN
					DP_Step1:=6666;
				END_IF
END_CASE
*)



*)
END_ACTION

ACTION _01Sticker_Auto:
TON_Sticker[4](PT:=T#200MS);//贴胶头夹紧气缸到位延时
rStickerStart_HMI(CLK:=Mach_Control.TJ_b.StickerStart_HMI , Q=> );
IF rStickerStart_HMI.Q THEN
	Sticker_SinStepMode:=FALSE;
END_IF
//贴胶自动程序
IF Mach_Control.U.TJ_iMode=1 OR AV THEN//在自动状态下
CASE Sticker_Step0 OF
		0://判断贴胶夹爪上是否有电芯，没电芯则移动至上电芯位，等待上电芯，有电芯则判断贴胶是否完成
				IF Mach_Control.TJ_b.StickerFlag THEN//判断贴胶夹爪上是否有电芯
						IF Mach_Control.TJ_b.StickerDone THEN//判断贴胶夹爪上的电芯是否贴胶完成
								Sticker_Step0:=1000;
						ELSIF NOT CellMemory[Mach_Control.TJ_b.TJ_Memory].Overhang_TF THEN//贴胶流程
								Sticker_Step0:=2000;
						ELSIF CellMemory[Mach_Control.TJ_b.TJ_Memory].Overhang_TF THEN//若是对齐度NG的料跳过贴胶流程										
								Mach_Control.TJ_b.StickerDone:=TRUE;//电芯贴胶完成
								Sticker_Step0:=0;							
						END_IF	
				ELSE
						Mach_Control.TJ_b.StickPermit:=FALSE;//贴胶允许
						Mach_Control.TJ_b.StickFinish:=FALSE;//贴胶完成	
						Mach_Control.TJ_b.StickMark_L1 :=FALSE;//左短边1贴胶完成
						Mach_Control.TJ_b.StickMark_L2 :=FALSE;//左短边2贴胶完成
 						Mach_Control.TJ_b.StickMark_R1 :=FALSE;//右短边1贴胶完成
						Mach_Control.TJ_b.StickMark_R2 :=FALSE;//右短边2贴胶完成		
						Mach_Control.TJ_b.StickMark1_L :=FALSE;//极耳侧贴胶完成		
						Mach_Control.TJ_b.StickMark1_L2 :=FALSE;//非极耳侧贴胶完成		
						Sticker_Step0:=100;
				END_IF	
		100:
			IF Mach_Control.WJ_b.TailCultOffloading AND NOT CellMemory[Mach_Control.TJ_b.TJ_Memory].Cell THEN
				Sticker_Step0:=150;
			ELSE
				Sticker_Step0:=0;
			END_IF
			
	
		150://允许侧贴胶平移、侧贴胶旋转动作 贴胶夹爪气缸张开，判断是否允许贴胶轴移动及旋转
				IF NOT Sticker_SinStepMode THEN			
						arrCyCtrl[arrCyNo.CylinderName.PullGlueModelCy].Cmd.bON:=TRUE;//贴胶冶具气缸打开
						
						IF 	 arrAxisCtrl[AxiseNo.AxisName.GluingWhirling].Status.Homed AND arrAxisCtrl[AxiseNo.AxisName.GluingWhirling].Status.NoMoving 
							AND arrCyCtrl[arrCyNo.CylinderName.PullGlueModelCy].Io.DIOnSwitch  AND Mach_Control.TJ_b.WhirlingSafe THEN
							IF arrAxisCtrl[AxiseNo.AxisName.GluingWhirling].Cmd.arrbRealPoint[5] THEN
								arrAxisCtrl[AxiseNo.AxisName.GluingWhirling].Cmd.iGoSetPos:=0;
							ELSE
								arrAxisCtrl[AxiseNo.AxisName.GluingWhirling].Cmd.iGoSetPos:=5;//侧贴胶夹旋转至上电芯位
							END_IF
						END_IF
						IF 	 arrAxisCtrl[AxiseNo.AxisName.GluingWhirling].Cmd.arrbRealPoint[5] AND arrCyCtrl[arrCyNo.CylinderName.PullGlueModelCy].Status.ONState THEN
							IF   Mach_Control.TJ_b.SinStepMode THEN//贴胶单步模式
								Sticker_SinStepMode:=TRUE;
							ELSE
								Sticker_SinStepMode:=FALSE;
							END_IF
							Sticker_Step0:=200;
						END_IF	
				END_IF			
		200:
			IF NOT Sticker_SinStepMode THEN			
					
					IF 	 arrAxisCtrl[AxiseNo.AxisName.GluingLine].Status.Homed AND arrAxisCtrl[AxiseNo.AxisName.GluingLine].Status.NoMoving AND
                       GluingLineagree  THEN
						IF arrAxisCtrl[AxiseNo.AxisName.GluingLine].Cmd.arrbRealPoint[8] THEN
							arrAxisCtrl[AxiseNo.AxisName.GluingLine].Cmd.iGoSetPos:=0;
						ELSE
							arrAxisCtrl[AxiseNo.AxisName.GluingLine].Cmd.iGoSetPos:=8;//侧贴胶夹平移至上电芯位
						END_IF
					END_IF	
					
					IF 	arrAxisCtrl[AxiseNo.AxisName.GluingLine].Cmd.arrbRealPoint[8]  THEN
						IF   Mach_Control.TJ_b.SinStepMode THEN//贴胶单步模式
							Sticker_SinStepMode:=TRUE;
						ELSE
							Sticker_SinStepMode:=FALSE;
						END_IF
						Sticker_Step0:=250;
					END_IF	
			END_IF			
		250:
				IF Mach_Control.TJ_b.StickerFlag AND arrAxisCtrl[AxiseNo.AxisName.TailCurlLine].Cmd.arrbRealPoint[10]
					AND arrAxisCtrl[AxiseNo.AxisName.TailCurlRetracting].Cmd.arrbRealPoint[1] 
					AND (arrCyCtrl[arrCyNo.CylinderName.PullGlueModelCy].Status.OFFState OR CellMemory[Mach_Control.TJ_b.TJ_Memory].Overhang_TF) THEN
						IF   Mach_Control.TJ_b.SinStepMode THEN//贴胶单步模式
								Sticker_SinStepMode:=TRUE;
						ELSE
								Sticker_SinStepMode:=FALSE;
						END_IF
							Sticker_Step0:=300;
				END_IF		
		300:
				IF NOT Sticker_SinStepMode THEN									
						IF 	 arrAxisCtrl[AxiseNo.AxisName.TailCurlRetracting].Cmd.arrbRealPoint[1] AND arrAxisCtrl[AxiseNo.AxisName.GluingLine].Status.Homed AND arrAxisCtrl[AxiseNo.AxisName.GluingLine].Status.NoMoving 
						AND Mach_Control.TJ_b.StickerFlag AND arrAxisCtrl[AxiseNo.AxisName.TailCurlLine].Cmd.arrbRealPoint[10]
					   AND arrAxisCtrl[AxiseNo.AxisName.TailCurlRetracting].Cmd.arrbRealPoint[1] AND GluingLineagree THEN
								IF arrAxisCtrl[AxiseNo.AxisName.GluingLine].Cmd.arrbRealPoint[1] THEN
									arrAxisCtrl[AxiseNo.AxisName.GluingLine].Cmd.iGoSetPos:=0;
								ELSE
									arrAxisCtrl[AxiseNo.AxisName.GluingLine].Cmd.iGoSetPos:=1;//侧贴胶夹平移至上极耳侧贴胶位
								END_IF
						END_IF	
						
						IF 	arrAxisCtrl[AxiseNo.AxisName.GluingLine].Cmd.arrbRealPoint[1]  THEN
								IF   Mach_Control.TJ_b.SinStepMode THEN//贴胶单步模式
										Sticker_SinStepMode:=TRUE;
								ELSE
										Sticker_SinStepMode:=FALSE;
								END_IF
							Sticker_Step0:=350;
						END_IF	
				END_IF			

		350:		
				IF NOT Sticker_SinStepMode THEN			
						IF 	arrAxisCtrl[AxiseNo.AxisName.GluingRetracting].Cmd.arrbRealPoint[1] AND arrAxisCtrl[AxiseNo.AxisName.GluingWhirling].Status.Homed 
							AND arrAxisCtrl[AxiseNo.AxisName.GluingWhirling].Status.NoMoving AND Mach_Control.TJ_b.WhirlingSafe THEN
								IF arrAxisCtrl[AxiseNo.AxisName.GluingWhirling].Cmd.arrbRealPoint[1] AND Mach_Control.TJ_b.StickerFlag AND arrAxisCtrl[AxiseNo.AxisName.TailCurlLine].Cmd.arrbRealPoint[10]
									AND arrAxisCtrl[AxiseNo.AxisName.TailCurlRetracting].Cmd.arrbRealPoint[1]   THEN
										arrAxisCtrl[AxiseNo.AxisName.GluingWhirling].Cmd.iGoSetPos:=0;
								ELSE
										arrAxisCtrl[AxiseNo.AxisName.GluingWhirling].Cmd.iGoSetPos:=1;//侧贴胶夹旋转至极耳侧贴胶位
								END_IF
						END_IF
						IF 	 arrAxisCtrl[AxiseNo.AxisName.GluingWhirling].Cmd.arrbRealPoint[1]  THEN
								IF   Mach_Control.TJ_b.SinStepMode THEN//贴胶单步模式
										Sticker_SinStepMode:=TRUE;
								ELSE
										Sticker_SinStepMode:=FALSE;
								END_IF
								Sticker_Step0:=400;
						END_IF	
				END_IF				
		400:
				IF NOT Sticker_SinStepMode THEN				
							Mach_Control.WJ_b.TailCultOffloading:=FALSE;//下电芯请求	
							//Mach_Control.TJ_b.StickerDone:=FALSE;//复位贴胶完成
							//Mach_Control.WJ_b.TailCultOffloadingDone:=FALSE;	
							IF Mach_Control.TJ_b.SinStepMode THEN//贴胶单步模式
									Sticker_SinStepMode:=TRUE;
							ELSE
									Sticker_SinStepMode:=FALSE;
							END_IF					
							Sticker_Step0:=0;		
				END_IF
				
				
		1000://贴胶完成，侧贴胶平移、侧贴胶旋转移动至下电芯位
				IF NOT Sticker_SinStepMode THEN		
						IF GluingLineagree AND arrAxisCtrl[AxiseNo.AxisName.GluingLine].Status.Homed AND arrAxisCtrl[AxiseNo.AxisName.GluingLine].Status.NoMoving   THEN
								IF arrAxisCtrl[AxiseNo.AxisName.GluingLine].Cmd.arrbRealPoint[9] THEN
										arrAxisCtrl[AxiseNo.AxisName.GluingLine].Cmd.iGoSetPos:=0;
								ELSE
										arrAxisCtrl[AxiseNo.AxisName.GluingLine].Cmd.iGoSetPos:=9;//侧贴胶夹平移至下电芯位
								END_IF
						END_IF	
						IF 	arrAxisCtrl[AxiseNo.AxisName.GluingWhirling].Status.Homed 
							AND arrAxisCtrl[AxiseNo.AxisName.GluingWhirling].Status.NoMoving AND Mach_Control.TJ_b.WhirlingSafe  THEN
								IF arrAxisCtrl[AxiseNo.AxisName.GluingWhirling].Cmd.arrbRealPoint[6] THEN
										arrAxisCtrl[AxiseNo.AxisName.GluingWhirling].Cmd.iGoSetPos:=0;
								ELSE
										arrAxisCtrl[AxiseNo.AxisName.GluingWhirling].Cmd.iGoSetPos:=6;//侧贴胶夹旋转至下电芯位
								END_IF
						END_IF
						IF 	arrAxisCtrl[AxiseNo.AxisName.GluingLine].Cmd.arrbRealPoint[9] AND arrAxisCtrl[AxiseNo.AxisName.GluingWhirling].Cmd.arrbRealPoint[6] THEN
								IF Mach_Control.TJ_b.SinStepMode THEN//贴胶单步模式
										Sticker_SinStepMode:=TRUE;
								ELSE
										Sticker_SinStepMode:=FALSE;
								END_IF						
								Sticker_Step0:=1100;
						END_IF	
				END_IF				
		//1100 信号交互挪到最下面
		
			1200://t贴胶旋转回原	
				Sticker_Step0:=1300;		
			1300:
				//arrCyCtrl[arrCyNo.CylinderName.GlueClampsCy].Cmd.bOFF:=TRUE;//贴胶夹爪气缸张开
				//IF 	arrCyCtrl[arrCyNo.CylinderName.GlueClampsCy].Io.DIOFFSwitch THEN
				IF Mach_Control.TJ_b.WhirlingSafe THEN
			     	arrAxisCtrl[AxiseNo.AxisName.GluingWhirling].Cmd.bHome:=TRUE;//侧贴胶旋转轴回原点
			    	Sticker_Step0:=1400;
				END_IF			
				//END_IF		
			1400://判断侧贴胶旋转回原是否完成
					StickerGohome_TON[4].IN:=TRUE;
					IF arrAxisCtrl[AxiseNo.AxisName.GluingWhirling].Status.Homed AND arrAxisCtrl[AxiseNo.AxisName.GluingWhirling].Status.NoMoving  AND StickerGohome_TON[4].Q THEN
						Sticker_Step0:=1500;
						arrAxisCtrl[AxiseNo.AxisName.GluingWhirling].Cmd.bHome:=FALSE;//侧贴胶旋转轴回原点
						StickerGohome_TON[4].IN:=FALSE;
					END_IF
			1500:	
				IF 	 arrAxisCtrl[AxiseNo.AxisName.GluingWhirling].Status.Homed AND arrAxisCtrl[AxiseNo.AxisName.GluingWhirling].Status.NoMoving AND Mach_Control.TJ_b.WhirlingSafe THEN
					IF arrAxisCtrl[AxiseNo.AxisName.GluingWhirling].Cmd.arrbRealPoint[5] THEN
						arrAxisCtrl[AxiseNo.AxisName.GluingWhirling].Cmd.iGoSetPos:=0;
						Sticker_Step0:=1600;
					ELSE
						arrAxisCtrl[AxiseNo.AxisName.GluingWhirling].Cmd.iGoSetPos:=5;//侧贴胶夹旋转至上电芯位
					END_IF
				END_IF
					
			1600:
				Sticker_Step0:=0;
				
		
				
				
				
		2000://判断贴胶状态
				IF  Mach_Control.TJ_b.StickMark_L1 AND   Mach_Control.TJ_b.StickMark_L2 AND   Mach_Control.TJ_b.StickMark_R1 AND   Mach_Control.TJ_b.StickMark_R2 AND  Mach_Control.TJ_b.StickMark1_L  AND (Mach_Control.TJ_b.StickMark1_L2 OR (NOT P3User2_Par.Shield[14] AND Sticker_Step2=0)) THEN
						Sticker_Step0:=5000;//贴胶完成
				ELSE
						IF NOT Mach_Control.TJ_b.StickMark_L1 THEN//左短边1贴胶完成
								Mach_Control.TJ_b.Sticking_L:=TRUE;//左短边贴胶
								Sticker_Step0:=2100;
						ELSIF NOT Mach_Control.TJ_b.StickMark_L2 THEN//左短边2贴胶完成
								Mach_Control.TJ_b.Sticking_L:=TRUE;//左短边贴胶
 								Sticker_Step0:=2600;
						ELSIF NOT Mach_Control.TJ_b.StickMark_R1 THEN//右短边1贴胶完成
								Mach_Control.TJ_b.Sticking_R:=TRUE;//右短边贴胶
								Sticker_Step0:=3100;
						ELSIF NOT Mach_Control.TJ_b.StickMark_R2 THEN//右短边2贴胶完成		
								Mach_Control.TJ_b.Sticking_R:=TRUE;//右短边贴胶
								Sticker_Step0:=3600;
						ELSIF NOT Mach_Control.TJ_b.StickMark1_L THEN//非极耳侧贴胶完成		
								Mach_Control.TJ_b.Sticking_Lg:=TRUE;//非极耳侧长边贴胶
								Sticker_Step0:=4100;
						ELSIF NOT Mach_Control.TJ_b.StickMark1_L2 AND  P3User2_Par.Shield[14] THEN//极耳侧贴胶完成		
								Mach_Control.TJ_b.Sticking_Lg2:=TRUE;//极耳侧长边贴胶
								Sticker_Step0:=4600;					
						END_IF
				END_IF
	
	
		2100://	左短边1贴胶
				IF NOT Sticker_SinStepMode THEN				
						arrCyCtrl[arrCyNo.CylinderName.GlueClampsCy].Cmd.bOFF:=TRUE;//贴胶夹爪气缸打开
						IF 	arrAxisCtrl[AxiseNo.AxisName.GluingLine].Status.Homed AND arrAxisCtrl[AxiseNo.AxisName.GluingLine].Status.NoMoving AND 
                           GluingLineagree THEN
							IF arrAxisCtrl[AxiseNo.AxisName.GluingLine].Cmd.arrbRealPoint[1] THEN
								arrAxisCtrl[AxiseNo.AxisName.GluingLine].Cmd.iGoSetPos:=0;
							ELSE
								arrAxisCtrl[AxiseNo.AxisName.GluingLine].Cmd.iGoSetPos:=1;//侧贴胶夹平移至贴胶位
							END_IF
						END_IF	
						IF 	arrAxisCtrl[AxiseNo.AxisName.GluingWhirling].Status.Homed AND arrAxisCtrl[AxiseNo.AxisName.GluingWhirling].Status.NoMoving AND Mach_Control.TJ_b.WhirlingSafe 
							AND 	arrAxisCtrl[AxiseNo.AxisName.GluingLine].Cmd.arrbRealPoint[1] THEN
							IF arrAxisCtrl[AxiseNo.AxisName.GluingWhirling].Cmd.arrbRealPoint[1] THEN
								arrAxisCtrl[AxiseNo.AxisName.GluingWhirling].Cmd.iGoSetPos:=0;
							ELSE
								arrAxisCtrl[AxiseNo.AxisName.GluingWhirling].Cmd.iGoSetPos:=1;//侧贴胶夹旋转至贴胶位
							END_IF
						END_IF
						IF 	arrAxisCtrl[AxiseNo.AxisName.GluingLine].Cmd.arrbRealPoint[1] AND arrAxisCtrl[AxiseNo.AxisName.GluingWhirling].Cmd.arrbRealPoint[1] 
							AND arrCyCtrl[arrCyNo.CylinderName.GlueClampsCy].Status.OFFState THEN
							IF Mach_Control.TJ_b.SinStepMode THEN//贴胶单眇模式
								Sticker_SinStepMode:=TRUE;
							ELSE
								Sticker_SinStepMode:=FALSE;
							END_IF										
							Sticker_Step0:=2200;
						END_IF
				END_IF		
		2200:
				Mach_Control.TJ_b.StickPermit:=TRUE;//贴胶允许
				Mach_Control.TJ_b.StickFinish:=FALSE;//贴胶完成			
				Sticker_Step0:=2300;
		2300:
				IF Mach_Control.TJ_b.StickFinish THEN//贴胶完成		
						Mach_Control.TJ_b.StickPermit:=FALSE;//贴胶允许	
						Sticker_Step0:=2400;
				END_IF 
		2400:
				Mach_Control.TJ_b.StickMark_L1:=TRUE;//左短边1贴胶完成
				Sticker_Step0:=2000;
				
		2600://	左短边2贴胶
				IF NOT Sticker_SinStepMode THEN				
						arrCyCtrl[arrCyNo.CylinderName.GlueClampsCy].Cmd.bOFF:=TRUE;//贴胶夹爪气缸打开
						IF 	arrAxisCtrl[AxiseNo.AxisName.GluingLine].Status.Homed AND arrAxisCtrl[AxiseNo.AxisName.GluingLine].Status.NoMoving AND GluingLineagree THEN
							IF arrAxisCtrl[AxiseNo.AxisName.GluingLine].Cmd.arrbRealPoint[2] THEN
								arrAxisCtrl[AxiseNo.AxisName.GluingLine].Cmd.iGoSetPos:=0;
							ELSE
								arrAxisCtrl[AxiseNo.AxisName.GluingLine].Cmd.iGoSetPos:=2;//侧贴胶夹平移至贴胶位
							END_IF
						END_IF	
						IF 	arrAxisCtrl[AxiseNo.AxisName.GluingWhirling].Status.Homed AND arrAxisCtrl[AxiseNo.AxisName.GluingWhirling].Status.NoMoving AND Mach_Control.TJ_b.WhirlingSafe  THEN
							IF arrAxisCtrl[AxiseNo.AxisName.GluingWhirling].Cmd.arrbRealPoint[1] THEN
								arrAxisCtrl[AxiseNo.AxisName.GluingWhirling].Cmd.iGoSetPos:=0;
							ELSE
								arrAxisCtrl[AxiseNo.AxisName.GluingWhirling].Cmd.iGoSetPos:=1;//侧贴胶夹旋转至贴胶位
							END_IF
						END_IF
						IF 	arrAxisCtrl[AxiseNo.AxisName.GluingLine].Cmd.arrbRealPoint[2] AND arrAxisCtrl[AxiseNo.AxisName.GluingWhirling].Cmd.arrbRealPoint[1] 
							AND arrCyCtrl[arrCyNo.CylinderName.GlueClampsCy].Status.OFFState THEN
							IF Mach_Control.TJ_b.SinStepMode THEN//贴胶单眇模式
								Sticker_SinStepMode:=TRUE;
							ELSE
								Sticker_SinStepMode:=FALSE;
							END_IF										
							Sticker_Step0:=2700;
						END_IF
				END_IF		
		2700:
				Mach_Control.TJ_b.StickPermit:=TRUE;//贴胶允许
				Mach_Control.TJ_b.StickFinish:=FALSE;//贴胶完成			
				Sticker_Step0:=2800;
		2800:
				IF Mach_Control.TJ_b.StickFinish THEN//贴胶完成		
						Mach_Control.TJ_b.StickPermit:=FALSE;//贴胶允许		
						Sticker_Step0:=2900;
				END_IF 
		2900:
				Mach_Control.TJ_b.StickMark_L2:=TRUE;//左短边2贴胶完成
				Sticker_Step0:=2000;
				
		3100://	右短边1贴胶
				IF NOT Sticker_SinStepMode THEN				
						arrCyCtrl[arrCyNo.CylinderName.GlueClampsCy].Cmd.bOFF:=TRUE;//贴胶夹爪气缸打开
						IF 	arrAxisCtrl[AxiseNo.AxisName.GluingLine].Status.Homed AND arrAxisCtrl[AxiseNo.AxisName.GluingLine].Status.NoMoving AND GluingLineagree THEN
							IF arrAxisCtrl[AxiseNo.AxisName.GluingLine].Cmd.arrbRealPoint[3] THEN
								arrAxisCtrl[AxiseNo.AxisName.GluingLine].Cmd.iGoSetPos:=0;
							ELSE
								arrAxisCtrl[AxiseNo.AxisName.GluingLine].Cmd.iGoSetPos:=3;//侧贴胶夹平移至贴胶位
							END_IF
						END_IF	
						IF 	arrAxisCtrl[AxiseNo.AxisName.GluingWhirling].Status.Homed AND arrAxisCtrl[AxiseNo.AxisName.GluingWhirling].Status.NoMoving AND Mach_Control.TJ_b.WhirlingSafe  THEN
							IF arrAxisCtrl[AxiseNo.AxisName.GluingWhirling].Cmd.arrbRealPoint[2] THEN
								arrAxisCtrl[AxiseNo.AxisName.GluingWhirling].Cmd.iGoSetPos:=0;
							ELSE
								arrAxisCtrl[AxiseNo.AxisName.GluingWhirling].Cmd.iGoSetPos:=2;//侧贴胶夹旋转至贴胶位2
							END_IF
						END_IF
						IF 	arrAxisCtrl[AxiseNo.AxisName.GluingLine].Cmd.arrbRealPoint[3] AND arrAxisCtrl[AxiseNo.AxisName.GluingWhirling].Cmd.arrbRealPoint[2] 
							AND arrCyCtrl[arrCyNo.CylinderName.GlueClampsCy].Status.OFFState THEN
							IF Mach_Control.TJ_b.SinStepMode THEN//贴胶单眇模式
								Sticker_SinStepMode:=TRUE;
							ELSE
								Sticker_SinStepMode:=FALSE;
							END_IF										
							Sticker_Step0:=3200;
						END_IF
				END_IF		
		3200:
				Mach_Control.TJ_b.StickPermit:=TRUE;//贴胶允许
				Mach_Control.TJ_b.StickFinish:=FALSE;//贴胶完成			
				Sticker_Step0:=3300;
		3300:
				IF Mach_Control.TJ_b.StickFinish THEN//贴胶完成			
						Mach_Control.TJ_b.StickPermit:=FALSE;//贴胶允许	
						Sticker_Step0:=3400;
				END_IF 
		3400:
				Mach_Control.TJ_b.StickMark_R1:=TRUE;//右短边1贴胶完成
				Sticker_Step0:=2000;
		
		
				
		3600://	右短边2贴胶
				IF NOT Sticker_SinStepMode THEN				
						arrCyCtrl[arrCyNo.CylinderName.GlueClampsCy].Cmd.bOFF:=TRUE;//贴胶夹爪气缸打开
						IF 	arrAxisCtrl[AxiseNo.AxisName.GluingLine].Status.Homed AND arrAxisCtrl[AxiseNo.AxisName.GluingLine].Status.NoMoving AND GluingLineagree THEN
								IF arrAxisCtrl[AxiseNo.AxisName.GluingLine].Cmd.arrbRealPoint[4] THEN
										arrAxisCtrl[AxiseNo.AxisName.GluingLine].Cmd.iGoSetPos:=0;
								ELSE
										arrAxisCtrl[AxiseNo.AxisName.GluingLine].Cmd.iGoSetPos:=4;//侧贴胶夹平移至贴胶位
								END_IF
						END_IF	
						IF 	arrAxisCtrl[AxiseNo.AxisName.GluingWhirling].Status.Homed AND arrAxisCtrl[AxiseNo.AxisName.GluingWhirling].Status.NoMoving AND Mach_Control.TJ_b.WhirlingSafe  THEN
								IF arrAxisCtrl[AxiseNo.AxisName.GluingWhirling].Cmd.arrbRealPoint[2] THEN
										arrAxisCtrl[AxiseNo.AxisName.GluingWhirling].Cmd.iGoSetPos:=0;
								ELSE
										arrAxisCtrl[AxiseNo.AxisName.GluingWhirling].Cmd.iGoSetPos:=2;//侧贴胶夹旋转至贴胶位2
								END_IF
						END_IF
						IF 	arrAxisCtrl[AxiseNo.AxisName.GluingLine].Cmd.arrbRealPoint[4] AND arrAxisCtrl[AxiseNo.AxisName.GluingWhirling].Cmd.arrbRealPoint[2] 
							AND arrCyCtrl[arrCyNo.CylinderName.GlueClampsCy].Status.OFFState THEN
								IF Mach_Control.TJ_b.SinStepMode THEN//贴胶单眇模式
										Sticker_SinStepMode:=TRUE;
								ELSE
										Sticker_SinStepMode:=FALSE;
								END_IF										
								Sticker_Step0:=3700;
						END_IF
				END_IF		
		3700:
				Mach_Control.TJ_b.StickPermit:=TRUE;//贴胶允许
				Mach_Control.TJ_b.StickFinish:=FALSE;//贴胶完成			
				Sticker_Step0:=3800;
		3800:
				IF Mach_Control.TJ_b.StickFinish THEN//贴胶完成			
						Mach_Control.TJ_b.StickPermit:=FALSE;//贴胶允许	
						Sticker_Step0:=3900;
				END_IF 
		3900:
				Mach_Control.TJ_b.StickMark_R2:=TRUE;//右短边1贴胶完成
				Sticker_Step0:=2000;
		

		4100://非极耳侧长边贴胶
			IF NOT Sticker_SinStepMode THEN				
						arrCyCtrl[arrCyNo.CylinderName.GlueClampsCy].Cmd.bOFF:=TRUE;//贴胶夹爪气缸打开
						IF 	arrAxisCtrl[AxiseNo.AxisName.GluingLine].Status.Homed AND arrAxisCtrl[AxiseNo.AxisName.GluingLine].Status.NoMoving AND GluingLineagree THEN
								IF arrAxisCtrl[AxiseNo.AxisName.GluingLine].Cmd.arrbRealPoint[5] THEN
										arrAxisCtrl[AxiseNo.AxisName.GluingLine].Cmd.iGoSetPos:=0;
								ELSE
										arrAxisCtrl[AxiseNo.AxisName.GluingLine].Cmd.iGoSetPos:=5;//侧贴胶夹平移至贴胶位
								END_IF
						END_IF	
						IF 	arrAxisCtrl[AxiseNo.AxisName.GluingWhirling].Status.Homed AND arrAxisCtrl[AxiseNo.AxisName.GluingWhirling].Status.NoMoving AND Mach_Control.TJ_b.WhirlingSafe  THEN
								IF arrAxisCtrl[AxiseNo.AxisName.GluingWhirling].Cmd.arrbRealPoint[3] THEN
										arrAxisCtrl[AxiseNo.AxisName.GluingWhirling].Cmd.iGoSetPos:=0;
								ELSE
										arrAxisCtrl[AxiseNo.AxisName.GluingWhirling].Cmd.iGoSetPos:=3;//侧贴胶夹旋转至贴胶位2
								END_IF
						END_IF
						IF 	arrAxisCtrl[AxiseNo.AxisName.GluingLine].Cmd.arrbRealPoint[5] AND arrAxisCtrl[AxiseNo.AxisName.GluingWhirling].Cmd.arrbRealPoint[3] 
							AND arrCyCtrl[arrCyNo.CylinderName.GlueClampsCy].Status.OFFState THEN
								IF Mach_Control.TJ_b.SinStepMode THEN//贴胶单眇模式
										Sticker_SinStepMode:=TRUE;
								ELSE
										Sticker_SinStepMode:=FALSE;
								END_IF										
								Sticker_Step0:=4200;
						END_IF
				END_IF		
		4200:
				Mach_Control.TJ_b.StickPermit:=TRUE;//贴胶允许
				Mach_Control.TJ_b.StickFinish:=FALSE;//贴胶完成			
				Sticker_Step0:=4300;
		4300:
				IF Mach_Control.TJ_b.StickFinish THEN//贴胶完成			
						Mach_Control.TJ_b.StickPermit:=FALSE;//贴胶允许	
						Sticker_Step0:=4400;
				END_IF 
		4400:
				Mach_Control.TJ_b.StickMark1_L:=TRUE;//非极耳侧长边贴胶完成
				Sticker_Step0:=2000;


		4600://极耳侧长边贴胶
			IF NOT Sticker_SinStepMode THEN				
						arrCyCtrl[arrCyNo.CylinderName.GlueClampsCy].Cmd.bOFF:=TRUE;//贴胶夹爪气缸打开
						IF 	arrAxisCtrl[AxiseNo.AxisName.GluingLine].Status.Homed AND arrAxisCtrl[AxiseNo.AxisName.GluingLine].Status.NoMoving AND GluingLineagree THEN
								IF arrAxisCtrl[AxiseNo.AxisName.GluingLine].Cmd.arrbRealPoint[6] THEN
										arrAxisCtrl[AxiseNo.AxisName.GluingLine].Cmd.iGoSetPos:=0;
								ELSE
										arrAxisCtrl[AxiseNo.AxisName.GluingLine].Cmd.iGoSetPos:=6;//侧贴胶夹平移至贴胶位
								END_IF
						END_IF	
						IF 	arrAxisCtrl[AxiseNo.AxisName.GluingWhirling].Status.Homed AND arrAxisCtrl[AxiseNo.AxisName.GluingWhirling].Status.NoMoving AND Mach_Control.TJ_b.WhirlingSafe  THEN
								IF arrAxisCtrl[AxiseNo.AxisName.GluingWhirling].Cmd.arrbRealPoint[4] THEN
										arrAxisCtrl[AxiseNo.AxisName.GluingWhirling].Cmd.iGoSetPos:=0;
								ELSE
										arrAxisCtrl[AxiseNo.AxisName.GluingWhirling].Cmd.iGoSetPos:=4;//侧贴胶夹旋转至贴胶位2
								END_IF
						END_IF
						IF 	arrAxisCtrl[AxiseNo.AxisName.GluingLine].Cmd.arrbRealPoint[6] AND arrAxisCtrl[AxiseNo.AxisName.GluingWhirling].Cmd.arrbRealPoint[4] 
							AND arrCyCtrl[arrCyNo.CylinderName.GlueClampsCy].Status.OFFState THEN
								IF Mach_Control.TJ_b.SinStepMode THEN//贴胶单眇模式
										Sticker_SinStepMode:=TRUE;
								ELSE
										Sticker_SinStepMode:=FALSE;
								END_IF										
								Sticker_Step0:=4700;
						END_IF
				END_IF		
		4700:
				Mach_Control.TJ_b.StickPermit:=TRUE;//贴胶允许
				Mach_Control.TJ_b.StickFinish:=FALSE;//贴胶完成			
				Sticker_Step0:=4800;
		4800:
				IF Mach_Control.TJ_b.StickFinish THEN//贴胶完成			
						Mach_Control.TJ_b.StickPermit:=FALSE;//贴胶允许	
						Sticker_Step0:=4900;
				END_IF 
		4900:
				Mach_Control.TJ_b.StickMark1_L2:=TRUE;//极耳侧长边贴胶完成
				Sticker_Step0:=2000;





	

	
		5000://等待贴胶完成信号						
				Mach_Control.TJ_b.StickerDone:=TRUE;//电芯贴胶完成
				CellMemory[Mach_Control.TJ_b.TJ_Memory].QR_code_No:=Par.stDT_date.QR_code_No;
				CellMemory[Mach_Control.TJ_b.TJ_Memory].Glue_No:=Par.stDT_date.Glue_No;		
				IF Mach_Control.TJ_b.SinStepMode THEN//贴胶单眇模式
					Sticker_SinStepMode:=TRUE;
				ELSE
					Sticker_SinStepMode:=FALSE;
				END_IF	
				Sticker_Step0:=5100;		
		5100:
				Mach_Control.TJ_b.StickPermit:=FALSE;//贴胶允许
				Mach_Control.TJ_b.StickFinish:=FALSE;//贴胶完成	
				Mach_Control.TJ_b.StickMark_L1 :=FALSE;//左短边1贴胶完成
				Mach_Control.TJ_b.StickMark_L2 :=FALSE;//左短边2贴胶完成
				Mach_Control.TJ_b.StickMark_R1 :=FALSE;//右短边1贴胶完成
				Mach_Control.TJ_b.StickMark_R2 :=FALSE;//右短边2贴胶完成	
				Mach_Control.TJ_b.StickMark1_L :=FALSE;//非极耳侧长边贴胶完成		
				Mach_Control.TJ_b.StickMark1_L2 :=FALSE;//极耳侧长边贴胶完成		
				Mach_Control.TJ_b.Sticking_L:=FALSE;//左短边贴胶
				Mach_Control.TJ_b.Sticking_R:=FALSE;//右短边贴胶
				Mach_Control.TJ_b.Sticking_Lg:=FALSE;//非极耳侧长边贴胶
				Mach_Control.TJ_b.Sticking_Lg2:=FALSE;//极耳侧长边贴胶
				Sticker_Step0:=0;		
				
				
END_CASE	
END_IF


